LIN {X 0,Y 566.204,Z 705.957,A -85,B 0,C 180,E1 -2372.429,E2 -2372.429} C_VEL
LIN {X 0,Y 566.171,Z 705.961,A -85,B 0,C 180,E1 -2374.988,E2 -2374.988} C_VEL
LIN {X 0,Y 566.186,Z 705.954,A -85,B 0,C 180,E1 -2377.462,E2 -2377.462} C_VEL
LIN {X 0,Y 566.206,Z 705.952,A -85,B 0,C 180,E1 -2380.199,E2 -2380.199} C_VEL
LIN {X 0,Y 566.18,Z 705.961,A -85,B 0,C 180,E1 -2383.057,E2 -2383.057} C_VEL
LIN {X 0,Y 566.158,Z 705.957,A -85,B 0,C 180,E1 -2386.053,E2 -2386.053} C_VEL
LIN {X 0,Y 566.151,Z 705.966,A -85,B 0,C 180,E1 -2388.858,E2 -2388.858} C_VEL
LIN {X 0,Y 566.201,Z 705.955,A -85,B 0,C 180,E1 -2391.444,E2 -2391.444} C_VEL
LIN {X 0,Y 566.139,Z 705.959,A -85,B 0,C 180,E1 -2394.306,E2 -2394.306} C_VEL
LIN {X 0,Y 566.163,Z 705.963,A -85,B 0,C 180,E1 -2396.894,E2 -2396.894} C_VEL
LIN {X 0,Y 566.16,Z 705.963,A -85,B 0,C 180,E1 -2399.406,E2 -2399.406} C_VEL
LIN {X 0,Y 566.149,Z 705.959,A -85,B 0,C 180,E1 -2401.854,E2 -2401.854} C_VEL
LIN {X 0,Y 566.168,Z 705.955,A -85,B 0,C 180,E1 -2404.249,E2 -2404.249} C_VEL
LIN {X 0,Y 566.164,Z 705.964,A -85,B 0,C 180,E1 -2407.368,E2 -2407.368} C_VEL
LIN {X 0,Y 566.203,Z 705.956,A -85,B 0,C 180,E1 -2409.662,E2 -2409.662} C_VEL
LIN {X 0,Y 566.167,Z 705.958,A -85,B 0,C 180,E1 -2411.921,E2 -2411.921} C_VEL
LIN {X 0,Y 566.183,Z 705.956,A -85,B 0,C 180,E1 -2414.89,E2 -2414.89} C_VEL
LIN {X 0,Y 566.18,Z 705.959,A -85,B 0,C 180,E1 -2417.818,E2 -2417.818} C_VEL
LIN {X 0,Y 566.136,Z 705.962,A -85,B 0,C 180,E1 -2419.991,E2 -2419.991} C_VEL
LIN {X 0,Y 566.185,Z 705.955,A -85,B 0,C 180,E1 -2422.152,E2 -2422.152} C_VEL
LIN {X 0,Y 566.257,Z 705.946,A -85,B 0,C 180,E1 -2425.016,E2 -2425.016} C_VEL
LIN {X 0,Y 566.277,Z 705.948,A -85,B 0,C 180,E1 -2427.866,E2 -2427.866} C_VEL
LIN {X 0,Y 566.288,Z 705.945,A -85,B 0,C 180,E1 -2430,E2 -2430} C_VEL
LIN {X 0,Y 566.245,Z 705.945,A -85,B 0,C 180,E1 -2432.846,E2 -2432.846} C_VEL
LIN {X 0,Y 566.244,Z 705.955,A -85,B 0,C 180,E1 -2435.699,E2 -2435.699} C_VEL
LIN {X 0,Y 566.201,Z 705.952,A -85,B 0,C 180,E1 -2438.566,E2 -2438.566} C_VEL
LIN {X 0,Y 566.244,Z 705.949,A -85,B 0,C 180,E1 -2441.454,E2 -2441.454} C_VEL
LIN {X 0,Y 566.238,Z 705.948,A -85,B 0,C 180,E1 -2444.506,E2 -2444.506} C_VEL
LIN {X 0,Y 566.193,Z 705.953,A -85,B 0,C 180,E1 -2447.332,E2 -2447.332} C_VEL
LIN {X 0,Y 566.209,Z 705.955,A -85,B 0,C 180,E1 -2450.338,E2 -2450.338} C_VEL
LIN {X 0,Y 566.171,Z 705.955,A -85,B 0,C 180,E1 -2453.28,E2 -2453.28} C_VEL
LIN {X 0,Y 566.196,Z 705.955,A -85,B 0,C 180,E1 -2455.75,E2 -2455.75} C_VEL
LIN {X 0,Y 566.189,Z 705.962,A -85,B 0,C 180,E1 -2458.199,E2 -2458.199} C_VEL
LIN {X 0,Y 566.191,Z 705.952,A -85,B 0,C 180,E1 -2461.076,E2 -2461.076} C_VEL
LIN {X 0,Y 566.201,Z 705.953,A -85,B 0,C 180,E1 -2463.732,E2 -2463.732} C_VEL
LIN {X 0,Y 566.204,Z 705.957,A -85,B 0,C 180,E1 -2466.57,E2 -2466.57} C_VEL
LIN {X 0,Y 566.218,Z 705.949,A -85,B 0,C 180,E1 -2469.686,E2 -2469.686} C_VEL
LIN {X 0,Y 566.206,Z 705.953,A -85,B 0,C 180,E1 -2472.917,E2 -2472.917} C_VEL
LIN {X 0,Y 566.198,Z 705.954,A -85,B 0,C 180,E1 -2476.049,E2 -2476.049} C_VEL
LIN {X 0,Y 566.208,Z 705.953,A -85,B 0,C 180,E1 -2479.215,E2 -2479.215} C_VEL
LIN {X 0,Y 566.23,Z 706.075,A -85,B 0,C 180,E1 -2479.979,E2 -2479.979} C_VEL
LIN {X 0,Y 566.747,Z 710.218,A -85,B 0,C 180,E1 -2480.146,E2 -2480.146} C_VEL
LIN {X 0,Y 566.638,Z 721.443,A -85,B 0,C 180,E1 -2480.667,E2 -2480.667} C_VEL
LIN {X 0,Y 566.488,Z 730.938,A -85,B 0,C 180,E1 -2481.217,E2 -2481.217} C_VEL
LIN {X 0,Y 566.359,Z 740.262,A -85,B 0,C 180,E1 -2481.877,E2 -2481.877} C_VEL
LIN {X 0,Y 566.256,Z 749.282,A -85,B 0,C 180,E1 -2482.649,E2 -2482.649} C_VEL
LIN {X 0,Y 566.168,Z 756.903,A -85,B 0,C 180,E1 -2483.427,E2 -2483.427} C_VEL
LIN {X 0,Y 566.072,Z 764.081,A -85,B 0,C 180,E1 -2484.301,E2 -2484.301} C_VEL
LIN {X 0,Y 566.051,Z 770.069,A -85,B 0,C 180,E1 -2485.171,E2 -2485.171} C_VEL
LIN {X 0,Y 565.969,Z 775.031,A -85,B 0,C 180,E1 -2486.027,E2 -2486.027} C_VEL
LIN {X 0,Y 565.906,Z 779.166,A -85,B 0,C 180,E1 -2486.877,E2 -2486.877} C_VEL
LIN {X 0,Y 565.892,Z 782.518,A -85,B 0,C 180,E1 -2487.722,E2 -2487.722} C_VEL
LIN {X 0,Y 565.881,Z 786.273,A -85,B 0,C 180,E1 -2488.976,E2 -2488.976} C_VEL
LIN {X 0,Y 565.882,Z 788.867,A -85,B 0,C 180,E1 -2490.386,E2 -2490.386} C_VEL
LIN {X 0,Y 565.848,Z 789.586,A -85,B 0,C 180,E1 -2491.027,E2 -2491.027} C_VEL
LIN {X 0,Y 565.846,Z 789.967,A -85,B 0,C 180,E1 -2491.866,E2 -2491.866} C_VEL
LIN {X 0,Y 565.833,Z 789.805,A -85,B 0,C 180,E1 -2492.641,E2 -2492.641} C_VEL
LIN {X 0,Y 565.862,Z 789.206,A -85,B 0,C 180,E1 -2493.441,E2 -2493.441} C_VEL
LIN {X 0,Y 565.839,Z 788.123,A -85,B 0,C 180,E1 -2494.232,E2 -2494.232} C_VEL
LIN {X 0,Y 565.914,Z 785.462,A -85,B 0,C 180,E1 -2495.428,E2 -2495.428} C_VEL
LIN {X 0,Y 565.913,Z 781.702,A -85,B 0,C 180,E1 -2496.584,E2 -2496.584} C_VEL
LIN {X 0,Y 565.935,Z 776.65,A -85,B 0,C 180,E1 -2497.743,E2 -2497.743} C_VEL
LIN {X 0,Y 565.996,Z 771.822,A -85,B 0,C 180,E1 -2498.636,E2 -2498.636} C_VEL
LIN {X 0,Y 566.072,Z 765.057,A -85,B 0,C 180,E1 -2499.657,E2 -2499.657} C_VEL
LIN {X 0,Y 566.15,Z 759.073,A -85,B 0,C 180,E1 -2500.417,E2 -2500.417} C_VEL
LIN {X 0,Y 566.234,Z 752.096,A -85,B 0,C 180,E1 -2501.173,E2 -2501.173} C_VEL
LIN {X 0,Y 566.338,Z 742.679,A -85,B 0,C 180,E1 -2502.02,E2 -2502.02} C_VEL
LIN {X 0,Y 566.436,Z 733.894,A -85,B 0,C 180,E1 -2502.676,E2 -2502.676} C_VEL
LIN {X 0,Y 566.533,Z 724.261,A -85,B 0,C 180,E1 -2503.27,E2 -2503.27} C_VEL
LIN {X 0,Y 566.663,Z 713.636,A -85,B 0,C 180,E1 -2503.796,E2 -2503.796} C_VEL
LIN {X 0,Y 566.73,Z 708.105,A -85,B 0,C 180,E1 -2504.029,E2 -2504.029} C_VEL
LIN {X 0,Y 566.222,Z 705.951,A -85,B 0,C 180,E1 -2504.13,E2 -2504.13} C_VEL
LIN {X 0,Y 566.196,Z 705.953,A -85,B 0,C 180,E1 -2506.359,E2 -2506.359} C_VEL
LIN {X 0,Y 566.24,Z 705.947,A -85,B 0,C 180,E1 -2508.675,E2 -2508.675} C_VEL
LIN {X 0,Y 566.227,Z 705.955,A -85,B 0,C 180,E1 -2511.434,E2 -2511.434} C_VEL
LIN {X 0,Y 566.251,Z 705.946,A -85,B 0,C 180,E1 -2514.302,E2 -2514.302} C_VEL
LIN {X 0,Y 566.284,Z 705.95,A -85,B 0,C 180,E1 -2517.866,E2 -2517.866} C_VEL
LIN {X 0,Y 566.303,Z 705.938,A -85,B 0,C 180,E1 -2520.711,E2 -2520.711} C_VEL
LIN {X 0,Y 566.273,Z 705.941,A -85,B 0,C 180,E1 -2522.845,E2 -2522.845} C_VEL
LIN {X 0,Y 566.256,Z 705.95,A -85,B 0,C 180,E1 -2525.698,E2 -2525.698} C_VEL
LIN {X 0,Y 566.224,Z 705.956,A -85,B 0,C 180,E1 -2527.847,E2 -2527.847} C_VEL
LIN {X 0,Y 566.243,Z 705.946,A -85,B 0,C 180,E1 -2530.73,E2 -2530.73} C_VEL
LIN {X 0,Y 566.21,Z 705.95,A -85,B 0,C 180,E1 -2532.91,E2 -2532.91} C_VEL
LIN {X 0,Y 566.203,Z 705.949,A -85,B 0,C 180,E1 -2535.109,E2 -2535.109} C_VEL
LIN {X 0,Y 566.204,Z 705.951,A -85,B 0,C 180,E1 -2537.332,E2 -2537.332} C_VEL
LIN {X 0,Y 566.212,Z 705.956,A -85,B 0,C 180,E1 -2540.337,E2 -2540.337} C_VEL
LIN {X 0,Y 566.173,Z 705.954,A -85,B 0,C 180,E1 -2543.281,E2 -2543.281} C_VEL
LIN {X 0,Y 566.213,Z 705.951,A -85,B 0,C 180,E1 -2545.749,E2 -2545.749} C_VEL
LIN {X 0,Y 566.207,Z 705.958,A -85,B 0,C 180,E1 -2548.202,E2 -2548.202} C_VEL
LIN {X 0,Y 566.195,Z 705.952,A -85,B 0,C 180,E1 -2551.076,E2 -2551.076} C_VEL
LIN {X 0,Y 566.216,Z 705.95,A -85,B 0,C 180,E1 -2553.734,E2 -2553.734} C_VEL
LIN {X 0,Y 566.204,Z 705.96,A -85,B 0,C 180,E1 -2556.57,E2 -2556.57} C_VEL
LIN {X 0,Y 566.225,Z 705.95,A -85,B 0,C 180,E1 -2559.273,E2 -2559.273} C_VEL
LIN {X 0,Y 566.193,Z 705.955,A -85,B 0,C 180,E1 -2562.089,E2 -2562.089} C_VEL
LIN {X 0,Y 566.177,Z 705.959,A -85,B 0,C 180,E1 -2565.036,E2 -2565.036} C_VEL
LIN {X 0,Y 566.222,Z 705.952,A -85,B 0,C 180,E1 -2568.136,E2 -2568.136} C_VEL
LIN {X 0,Y 566.219,Z 705.96,A -85,B 0,C 180,E1 -2570.726,E2 -2570.726} C_VEL
LIN {X 0,Y 566.241,Z 706.07,A -85,B 0,C 180,E1 -2572.989,E2 -2572.989} C_VEL
LIN {X 0,Y 567.262,Z 712.594,A -85,B 0,C 180,E1 -2574.387,E2 -2574.387} C_VEL
LIN {X 0,Y 567.322,Z 727.831,A -85,B 0,C 180,E1 -2577.393,E2 -2577.393} C_VEL
LIN {X 0,Y 567.311,Z 742.969,A -85,B 0,C 180,E1 -2580.295,E2 -2580.295} C_VEL
LIN {X 0,Y 567.031,Z 758.624,A -85,B 0,C 180,E1 -2583.5,E2 -2583.5} C_VEL
LIN {X 0,Y 566.812,Z 772.321,A -85,B 0,C 180,E1 -2586.236,E2 -2586.236} C_VEL
LIN {X 0,Y 566.605,Z 787.97,A -85,B 0,C 180,E1 -2589.298,E2 -2589.298} C_VEL
LIN {X 0,Y 566.401,Z 803.622,A -85,B 0,C 180,E1 -2592.302,E2 -2592.302} C_VEL
LIN {X 0,Y 566.238,Z 819.258,A -85,B 0,C 180,E1 -2595.256,E2 -2595.256} C_VEL
LIN {X 0,Y 566.153,Z 830.11,A -85,B 0,C 180,E1 -2597.285,E2 -2597.285} C_VEL
LIN {X 0,Y 566.954,Z 837.081,A -85,B 0,C 180,E1 -2597.426,E2 -2597.426} C_VEL
LIN {X 0,Y 566.844,Z 850.733,A -85,B 0,C 180,E1 -2597.764,E2 -2597.764} C_VEL
LIN {X 0,Y 566.707,Z 863.522,A -85,B 0,C 180,E1 -2598.238,E2 -2598.238} C_VEL
LIN {X 0,Y 566.572,Z 875.723,A -85,B 0,C 180,E1 -2598.854,E2 -2598.854} C_VEL
LIN {X 0,Y 566.421,Z 886.478,A -85,B 0,C 180,E1 -2599.545,E2 -2599.545} C_VEL
LIN {X 0,Y 566.297,Z 896.645,A -85,B 0,C 180,E1 -2600.355,E2 -2600.355} C_VEL
LIN {X 0,Y 566.166,Z 905.786,A -85,B 0,C 180,E1 -2601.253,E2 -2601.253} C_VEL
LIN {X 0,Y 566.081,Z 914.689,A -85,B 0,C 180,E1 -2602.33,E2 -2602.33} C_VEL
LIN {X 0,Y 565.967,Z 921.955,A -85,B 0,C 180,E1 -2603.422,E2 -2603.422} C_VEL
LIN {X 0,Y 566.004,Z 926.68,A -85,B 0,C 180,E1 -2604.299,E2 -2604.299} C_VEL
LIN {X 0,Y 565.933,Z 931.371,A -85,B 0,C 180,E1 -2605.37,E2 -2605.37} C_VEL
LIN {X 0,Y 565.927,Z 934.957,A -85,B 0,C 180,E1 -2606.44,E2 -2606.44} C_VEL
LIN {X 0,Y 565.878,Z 936.808,A -85,B 0,C 180,E1 -2607.152,E2 -2607.152} C_VEL
LIN {X 0,Y 565.838,Z 938.199,A -85,B 0,C 180,E1 -2607.864,E2 -2607.864} C_VEL
LIN {X 0,Y 565.841,Z 939.785,A -85,B 0,C 180,E1 -2609.288,E2 -2609.288} C_VEL
LIN {X 0,Y 565.839,Z 940,A -85,B 0,C 180,E1 -2610,E2 -2610} C_VEL
LIN {X 0,Y 565.846,Z 939.186,A -85,B 0,C 180,E1 -2611.423,E2 -2611.423} C_VEL
LIN {X 0,Y 565.838,Z 938.2,A -85,B 0,C 180,E1 -2612.135,E2 -2612.135} C_VEL
LIN {X 0,Y 565.878,Z 936.81,A -85,B 0,C 180,E1 -2612.847,E2 -2612.847} C_VEL
LIN {X 0,Y 565.926,Z 933.896,A -85,B 0,C 180,E1 -2613.916,E2 -2613.916} C_VEL
LIN {X 0,Y 565.878,Z 929.949,A -85,B 0,C 180,E1 -2614.987,E2 -2614.987} C_VEL
LIN {X 0,Y 566.002,Z 924.867,A -85,B 0,C 180,E1 -2616.058,E2 -2616.058} C_VEL
LIN {X 0,Y 566.04,Z 918.469,A -85,B 0,C 180,E1 -2617.132,E2 -2617.132} C_VEL
LIN {X 0,Y 566.133,Z 910.479,A -85,B 0,C 180,E1 -2618.208,E2 -2618.208} C_VEL
LIN {X 0,Y 566.229,Z 902.337,A -85,B 0,C 180,E1 -2619.105,E2 -2619.105} C_VEL
LIN {X 0,Y 566.34,Z 892.402,A -85,B 0,C 180,E1 -2620.005,E2 -2620.005} C_VEL
LIN {X 0,Y 566.536,Z 881.306,A -85,B 0,C 180,E1 -2620.806,E2 -2620.806} C_VEL
LIN {X 0,Y 566.613,Z 870.179,A -85,B 0,C 180,E1 -2621.447,E2 -2621.447} C_VEL
LIN {X 0,Y 566.742,Z 857.987,A -85,B 0,C 180,E1 -2621.988,E2 -2621.988} C_VEL
LIN {X 0,Y 566.913,Z 845.178,A -85,B 0,C 180,E1 -2622.393,E2 -2622.393} C_VEL
LIN {X 0,Y 566.761,Z 833.946,A -85,B 0,C 180,E1 -2622.634,E2 -2622.634} C_VEL
LIN {X 0,Y 566.154,Z 830.034,A -85,B 0,C 180,E1 -2622.729,E2 -2622.729} C_VEL
LIN {X 0,Y 566.282,Z 815.361,A -85,B 0,C 180,E1 -2625.476,E2 -2625.476} C_VEL
LIN {X 0,Y 566.456,Z 799.71,A -85,B 0,C 180,E1 -2628.444,E2 -2628.444} C_VEL
LIN {X 0,Y 566.62,Z 784.878,A -85,B 0,C 180,E1 -2631.303,E2 -2631.303} C_VEL
LIN {X 0,Y 566.836,Z 770.363,A -85,B 0,C 180,E1 -2634.152,E2 -2634.152} C_VEL
LIN {X 0,Y 567.064,Z 756.117,A -85,B 0,C 180,E1 -2637.008,E2 -2637.008} C_VEL
LIN {X 0,Y 567.313,Z 742.161,A -85,B 0,C 180,E1 -2639.868,E2 -2639.868} C_VEL
LIN {X 0,Y 567.407,Z 727.53,A -85,B 0,C 180,E1 -2642.775,E2 -2642.775} C_VEL
LIN {X 0,Y 567.477,Z 715.115,A -85,B 0,C 180,E1 -2645.334,E2 -2645.334} C_VEL
LIN {X 0,Y 567.176,Z 710.471,A -85,B 0,C 180,E1 -2646.348,E2 -2646.348} C_VEL
LIN {X 0,Y 566.203,Z 705.96,A -85,B 0,C 180,E1 -2647.401,E2 -2647.401} C_VEL
LIN {X 0,Y 566.22,Z 705.951,A -85,B 0,C 180,E1 -2650.198,E2 -2650.198} C_VEL
LIN {X 0,Y 566.205,Z 705.958,A -85,B 0,C 180,E1 -2653.054,E2 -2653.054} C_VEL
LIN {X 0,Y 566.201,Z 705.952,A -85,B 0,C 180,E1 -2656.049,E2 -2656.049} C_VEL
LIN {X 0,Y 566.223,Z 705.956,A -85,B 0,C 180,E1 -2659.213,E2 -2659.213} C_VEL
LIN {X 0,Y 566.192,Z 705.959,A -85,B 0,C 180,E1 -2661.637,E2 -2661.637} C_VEL
LIN {X 0,Y 566.168,Z 705.955,A -85,B 0,C 180,E1 -2664.308,E2 -2664.308} C_VEL
LIN {X 0,Y 566.232,Z 705.948,A -85,B 0,C 180,E1 -2666.899,E2 -2666.899} C_VEL
LIN {X 0,Y 566.184,Z 705.96,A -85,B 0,C 180,E1 -2669.407,E2 -2669.407} C_VEL
LIN {X 0,Y 566.215,Z 705.955,A -85,B 0,C 180,E1 -2671.857,E2 -2671.857} C_VEL
LIN {X 0,Y 566.215,Z 705.951,A -85,B 0,C 180,E1 -2674.251,E2 -2674.251} C_VEL
LIN {X 0,Y 566.172,Z 705.954,A -85,B 0,C 180,E1 -2676.719,E2 -2676.719} C_VEL
LIN {X 0,Y 566.211,Z 705.958,A -85,B 0,C 180,E1 -2679.663,E2 -2679.663} C_VEL
LIN {X 0,Y 566.202,Z 705.951,A -85,B 0,C 180,E1 -2682.668,E2 -2682.668} C_VEL
LIN {X 0,Y 566.236,Z 705.953,A -85,B 0,C 180,E1 -2685.627,E2 -2685.627} C_VEL
LIN {X 0,Y 566.239,Z 705.947,A -85,B 0,C 180,E1 -2688.675,E2 -2688.675} C_VEL
LIN {X 0,Y 566.229,Z 705.95,A -85,B 0,C 180,E1 -2691.434,E2 -2691.434} C_VEL
LIN {X 0,Y 566.252,Z 705.95,A -85,B 0,C 180,E1 -2694.302,E2 -2694.302} C_VEL
LIN {X 0,Y 566.286,Z 705.947,A -85,B 0,C 180,E1 -2697.866,E2 -2697.866} C_VEL
LIN {X 0,Y 566.292,Z 705.941,A -85,B 0,C 180,E1 -2700.711,E2 -2700.711} C_VEL
LIN {X 0,Y 566.261,Z 705.945,A -85,B 0,C 180,E1 -2702.846,E2 -2702.846} C_VEL
LIN {X 0,Y 566.249,Z 705.948,A -85,B 0,C 180,E1 -2705.699,E2 -2705.699} C_VEL
LIN {X 0,Y 566.225,Z 705.953,A -85,B 0,C 180,E1 -2708.566,E2 -2708.566} C_VEL
LIN {X 0,Y 566.245,Z 705.946,A -85,B 0,C 180,E1 -2711.454,E2 -2711.454} C_VEL
LIN {X 0,Y 566.225,Z 705.956,A -85,B 0,C 180,E1 -2714.502,E2 -2714.502} C_VEL
LIN {X 0,Y 566.191,Z 705.952,A -85,B 0,C 180,E1 -2717.332,E2 -2717.332} C_VEL
LIN {X 0,Y 566.204,Z 705.951,A -85,B 0,C 180,E1 -2719.581,E2 -2719.581} C_VEL
LIN {X 0,Y 566.193,Z 705.953,A -85,B 0,C 180,E1 -2721.863,E2 -2721.863} C_VEL
LIN {X 0,Y 566.181,Z 705.957,A -85,B 0,C 180,E1 -2725.021,E2 -2725.021} C_VEL
LIN {X 0,Y 566.163,Z 705.956,A -85,B 0,C 180,E1 -2727.461,E2 -2727.461} C_VEL
LIN {X 0,Y 565.494,Z 706.042,A -85,B 0,C 180,E1 -2728.055,E2 -2728.055} C_VEL
LIN {X 0,Y 562.638,Z 706.399,A -85,B 0,C 180,E1 -2729.019,E2 -2729.019} C_VEL
LIN {X 0,Y 560.231,Z 706.698,A -85,B 0,C 180,E1 -2729.795,E2 -2729.795} C_VEL
LIN {X 0,Y 559.207,Z 706.829,A -85,B 0,C 180,E1 -2730.393,E2 -2730.393} C_VEL
LIN {X 0,Y 559.129,Z 706.834,A -85,B 0,C 180,E1 -2730.596,E2 -2730.596} C_VEL
LIN {X 0,Y 559.153,Z 706.838,A -85,B 0,C 180,E1 -2732.716,E2 -2732.716} C_VEL
LIN {X 0,Y 559.12,Z 706.835,A -85,B 0,C 180,E1 -2735.325,E2 -2735.325} C_VEL
LIN {X 0,Y 559.124,Z 706.833,A -85,B 0,C 180,E1 -2738.019,E2 -2738.019} C_VEL
LIN {X 0,Y 559.127,Z 706.841,A -85,B 0,C 180,E1 -2740.815,E2 -2740.815} C_VEL
LIN {X 0,Y 559.108,Z 706.835,A -85,B 0,C 180,E1 -2743.738,E2 -2743.738} C_VEL
LIN {X 0,Y 559.109,Z 706.836,A -85,B 0,C 180,E1 -2746.263,E2 -2746.263} C_VEL
LIN {X 0,Y 559.116,Z 706.841,A -85,B 0,C 180,E1 -2749.184,E2 -2749.184} C_VEL
LIN {X 0,Y 559.169,Z 706.835,A -85,B 0,C 180,E1 -2751.193,E2 -2751.193} C_VEL
LIN {X 0,Y 559.115,Z 706.835,A -85,B 0,C 180,E1 -2753.787,E2 -2753.787} C_VEL
LIN {X 0,Y 559.125,Z 706.834,A -85,B 0,C 180,E1 -2756.422,E2 -2756.422} C_VEL
LIN {X 0,Y 559.143,Z 706.838,A -85,B 0,C 180,E1 -2758.98,E2 -2758.98} C_VEL
LIN {X 0,Y 559.11,Z 706.838,A -85,B 0,C 180,E1 -2761.631,E2 -2761.631} C_VEL
LIN {X 0,Y 559.115,Z 706.835,A -85,B 0,C 180,E1 -2763.9,E2 -2763.9} C_VEL
LIN {X 0,Y 559.114,Z 706.841,A -85,B 0,C 180,E1 -2767.066,E2 -2767.066} C_VEL
LIN {X 0,Y 559.174,Z 706.835,A -85,B 0,C 180,E1 -2769.395,E2 -2769.395} C_VEL
LIN {X 0,Y 559.119,Z 706.839,A -85,B 0,C 180,E1 -2771.685,E2 -2771.685} C_VEL
LIN {X 0,Y 559.139,Z 706.833,A -85,B 0,C 180,E1 -2773.947,E2 -2773.947} C_VEL
LIN {X 0,Y 559.146,Z 706.831,A -85,B 0,C 180,E1 -2776.183,E2 -2776.183} C_VEL
LIN {X 0,Y 559.158,Z 706.833,A -85,B 0,C 180,E1 -2779.133,E2 -2779.133} C_VEL
LIN {X 0,Y 559.139,Z 706.834,A -85,B 0,C 180,E1 -2782.053,E2 -2782.053} C_VEL
LIN {X 0,Y 559.232,Z 706.821,A -85,B 0,C 180,E1 -2784.953,E2 -2784.953} C_VEL
LIN {X 0,Y 559.248,Z 706.824,A -85,B 0,C 180,E1 -2787.839,E2 -2787.839} C_VEL
LIN {X 0,Y 559.257,Z 706.821,A -85,B 0,C 180,E1 -2790,E2 -2790} C_VEL
LIN {X 0,Y 559.213,Z 706.822,A -85,B 0,C 180,E1 -2792.882,E2 -2792.882} C_VEL
LIN {X 0,Y 559.214,Z 706.831,A -85,B 0,C 180,E1 -2795.77,E2 -2795.77} C_VEL
LIN {X 0,Y 559.166,Z 706.828,A -85,B 0,C 180,E1 -2798.675,E2 -2798.675} C_VEL
LIN {X 0,Y 559.206,Z 706.828,A -85,B 0,C 180,E1 -2801.601,E2 -2801.601} C_VEL
LIN {X 0,Y 559.206,Z 706.824,A -85,B 0,C 180,E1 -2804.596,E2 -2804.596} C_VEL
LIN {X 0,Y 559.138,Z 706.834,A -85,B 0,C 180,E1 -2807.558,E2 -2807.558} C_VEL
LIN {X 0,Y 559.169,Z 706.834,A -85,B 0,C 180,E1 -2809.838,E2 -2809.838} C_VEL
LIN {X 0,Y 559.143,Z 706.839,A -85,B 0,C 180,E1 -2812.153,E2 -2812.153} C_VEL
LIN {X 0,Y 559.145,Z 706.83,A -85,B 0,C 180,E1 -2815.178,E2 -2815.178} C_VEL
LIN {X 0,Y 559.129,Z 706.835,A -85,B 0,C 180,E1 -2817.715,E2 -2817.715} C_VEL
LIN {X 0,Y 559.153,Z 706.839,A -85,B 0,C 180,E1 -2820.183,E2 -2820.183} C_VEL
LIN {X 0,Y 559.155,Z 706.832,A -85,B 0,C 180,E1 -2822.716,E2 -2822.716} C_VEL
LIN {X 0,Y 559.131,Z 706.831,A -85,B 0,C 180,E1 -2825.324,E2 -2825.324} C_VEL
LIN {X 0,Y 559.137,Z 706.835,A -85,B 0,C 180,E1 -2828.018,E2 -2828.018} C_VEL
LIN {X 0,Y 559.159,Z 706.831,A -85,B 0,C 180,E1 -2830.813,E2 -2830.813} C_VEL
LIN {X 0,Y 559.142,Z 706.83,A -85,B 0,C 180,E1 -2833.734,E2 -2833.734} C_VEL
LIN {X 0,Y 559.149,Z 706.836,A -85,B 0,C 180,E1 -2836.804,E2 -2836.804} C_VEL
LIN {X 0,Y 559.177,Z 706.829,A -85,B 0,C 180,E1 -2839.837,E2 -2839.837} C_VEL
LIN {X 0,Y 559.788,Z 710.922,A -85,B 0,C 180,E1 -2840.028,E2 -2840.028} C_VEL
LIN {X 0,Y 559.658,Z 721.465,A -85,B 0,C 180,E1 -2840.525,E2 -2840.525} C_VEL
LIN {X 0,Y 559.472,Z 732.021,A -85,B 0,C 180,E1 -2841.154,E2 -2841.154} C_VEL
LIN {X 0,Y 559.336,Z 740.517,A -85,B 0,C 180,E1 -2841.77,E2 -2841.77} C_VEL
LIN {X 0,Y 559.236,Z 748.955,A -85,B 0,C 180,E1 -2842.499,E2 -2842.499} C_VEL
LIN {X 0,Y 559.108,Z 756.352,A -85,B 0,C 180,E1 -2843.256,E2 -2843.256} C_VEL
LIN {X 0,Y 559.03,Z 762.612,A -85,B 0,C 180,E1 -2844.004,E2 -2844.004} C_VEL
LIN {X 0,Y 558.956,Z 769.522,A -85,B 0,C 180,E1 -2844.995,E2 -2844.995} C_VEL
LIN {X 0,Y 558.891,Z 774.491,A -85,B 0,C 180,E1 -2845.844,E2 -2845.844} C_VEL
LIN {X 0,Y 558.842,Z 779.251,A -85,B 0,C 180,E1 -2846.834,E2 -2846.834} C_VEL
LIN {X 0,Y 558.796,Z 783.939,A -85,B 0,C 180,E1 -2848.113,E2 -2848.113} C_VEL
LIN {X 0,Y 558.783,Z 786.313,A -85,B 0,C 180,E1 -2848.957,E2 -2848.957} C_VEL
LIN {X 0,Y 558.774,Z 788.662,A -85,B 0,C 180,E1 -2850.21,E2 -2850.21} C_VEL
LIN {X 0,Y 558.75,Z 789.905,A -85,B 0,C 180,E1 -2851.699,E2 -2851.699} C_VEL
LIN {X 0,Y 558.75,Z 789.585,A -85,B 0,C 180,E1 -2853.076,E2 -2853.076} C_VEL
LIN {X 0,Y 558.742,Z 788.659,A -85,B 0,C 180,E1 -2853.881,E2 -2853.881} C_VEL
LIN {X 0,Y 558.783,Z 786.806,A -85,B 0,C 180,E1 -2854.901,E2 -2854.901} C_VEL
LIN {X 0,Y 558.807,Z 784.25,A -85,B 0,C 180,E1 -2855.874,E2 -2855.874} C_VEL
LIN {X 0,Y 558.821,Z 780.058,A -85,B 0,C 180,E1 -2857.053,E2 -2857.053} C_VEL
LIN {X 0,Y 558.888,Z 774.655,A -85,B 0,C 180,E1 -2858.213,E2 -2858.213} C_VEL
LIN {X 0,Y 558.981,Z 767.676,A -85,B 0,C 180,E1 -2859.388,E2 -2859.388} C_VEL
LIN {X 0,Y 559.108,Z 759.09,A -85,B 0,C 180,E1 -2860.52,E2 -2860.52} C_VEL
LIN {X 0,Y 559.193,Z 751.891,A -85,B 0,C 180,E1 -2861.307,E2 -2861.307} C_VEL
LIN {X 0,Y 559.324,Z 743.595,A -85,B 0,C 180,E1 -2862.07,E2 -2862.07} C_VEL
LIN {X 0,Y 559.446,Z 733.913,A -85,B 0,C 180,E1 -2862.807,E2 -2862.807} C_VEL
LIN {X 0,Y 559.55,Z 724.513,A -85,B 0,C 180,E1 -2863.397,E2 -2863.397} C_VEL
LIN {X 0,Y 559.668,Z 715.312,A -85,B 0,C 180,E1 -2863.869,E2 -2863.869} C_VEL
LIN {X 0,Y 559.647,Z 708.978,A -85,B 0,C 180,E1 -2864.149,E2 -2864.149} C_VEL
LIN {X 0,Y 559.169,Z 706.83,A -85,B 0,C 180,E1 -2864.252,E2 -2864.252} C_VEL
LIN {X 0,Y 559.162,Z 706.83,A -85,B 0,C 180,E1 -2866.924,E2 -2866.924} C_VEL
LIN {X 0,Y 559.197,Z 706.828,A -85,B 0,C 180,E1 -2869.133,E2 -2869.133} C_VEL
LIN {X 0,Y 559.202,Z 706.827,A -85,B 0,C 180,E1 -2872.053,E2 -2872.053} C_VEL
LIN {X 0,Y 559.245,Z 706.818,A -85,B 0,C 180,E1 -2874.953,E2 -2874.953} C_VEL
LIN {X 0,Y 559.255,Z 706.826,A -85,B 0,C 180,E1 -2877.839,E2 -2877.839} C_VEL
LIN {X 0,Y 559.273,Z 706.814,A -85,B 0,C 180,E1 -2880.72,E2 -2880.72} C_VEL
LIN {X 0,Y 559.239,Z 706.817,A -85,B 0,C 180,E1 -2882.881,E2 -2882.881} C_VEL
LIN {X 0,Y 559.226,Z 706.827,A -85,B 0,C 180,E1 -2885.77,E2 -2885.77} C_VEL
LIN {X 0,Y 559.174,Z 706.826,A -85,B 0,C 180,E1 -2888.675,E2 -2888.675} C_VEL
LIN {X 0,Y 559.21,Z 706.825,A -85,B 0,C 180,E1 -2891.6,E2 -2891.6} C_VEL
LIN {X 0,Y 559.205,Z 706.823,A -85,B 0,C 180,E1 -2894.595,E2 -2894.595} C_VEL
LIN {X 0,Y 559.147,Z 706.831,A -85,B 0,C 180,E1 -2897.557,E2 -2897.557} C_VEL
LIN {X 0,Y 559.171,Z 706.831,A -85,B 0,C 180,E1 -2899.837,E2 -2899.837} C_VEL
LIN {X 0,Y 559.145,Z 706.838,A -85,B 0,C 180,E1 -2902.153,E2 -2902.153} C_VEL
LIN {X 0,Y 559.179,Z 706.826,A -85,B 0,C 180,E1 -2905.298,E2 -2905.298} C_VEL
LIN {X 0,Y 559.161,Z 706.829,A -85,B 0,C 180,E1 -2907.713,E2 -2907.713} C_VEL
LIN {X 0,Y 559.157,Z 706.835,A -85,B 0,C 180,E1 -2910.183,E2 -2910.183} C_VEL
LIN {X 0,Y 559.179,Z 706.831,A -85,B 0,C 180,E1 -2912.714,E2 -2912.714} C_VEL
LIN {X 0,Y 559.134,Z 706.832,A -85,B 0,C 180,E1 -2915.324,E2 -2915.324} C_VEL
LIN {X 0,Y 559.138,Z 706.834,A -85,B 0,C 180,E1 -2918.017,E2 -2918.017} C_VEL
LIN {X 0,Y 559.177,Z 706.833,A -85,B 0,C 180,E1 -2920.811,E2 -2920.811} C_VEL
LIN {X 0,Y 559.145,Z 706.831,A -85,B 0,C 180,E1 -2923.734,E2 -2923.734} C_VEL
LIN {X 0,Y 559.169,Z 706.837,A -85,B 0,C 180,E1 -2926.801,E2 -2926.801} C_VEL
LIN {X 0,Y 559.166,Z 706.835,A -85,B 0,C 180,E1 -2929.188,E2 -2929.188} C_VEL
LIN {X 0,Y 559.137,Z 706.837,A -85,B 0,C 180,E1 -2931.982,E2 -2931.982} C_VEL
LIN {X 0,Y 559.198,Z 706.945,A -85,B 0,C 180,E1 -2932.798,E2 -2932.798} C_VEL
LIN {X 0,Y 560.308,Z 713.782,A -85,B 0,C 180,E1 -2934.287,E2 -2934.287} C_VEL
LIN {X 0,Y 560.332,Z 729.084,A -85,B 0,C 180,E1 -2937.362,E2 -2937.362} C_VEL
LIN {X 0,Y 560.32,Z 743.41,A -85,B 0,C 180,E1 -2940.13,E2 -2940.13} C_VEL
LIN {X 0,Y 560.217,Z 752.754,A -85,B 0,C 180,E1 -2941.937,E2 -2941.937} C_VEL
LIN {X 0,Y 559.994,Z 766.449,A -85,B 0,C 180,E1 -2944.741,E2 -2944.741} C_VEL
LIN {X 0,Y 559.741,Z 780.144,A -85,B 0,C 180,E1 -2947.483,E2 -2947.483} C_VEL
LIN {X 0,Y 559.514,Z 795.003,A -85,B 0,C 180,E1 -2950.402,E2 -2950.402} C_VEL
LIN {X 0,Y 559.329,Z 809.491,A -85,B 0,C 180,E1 -2953.202,E2 -2953.202} C_VEL
LIN {X 0,Y 559.173,Z 825.142,A -85,B 0,C 180,E1 -2956.184,E2 -2956.184} C_VEL
LIN {X 0,Y 559.103,Z 830.156,A -85,B 0,C 180,E1 -2957.131,E2 -2957.131} C_VEL
LIN {X 0,Y 560.027,Z 837.081,A -85,B 0,C 180,E1 -2957.267,E2 -2957.267} C_VEL
LIN {X 0,Y 559.91,Z 850.734,A -85,B 0,C 180,E1 -2957.61,E2 -2957.61} C_VEL
LIN {X 0,Y 559.77,Z 863.521,A -85,B 0,C 180,E1 -2958.09,E2 -2958.09} C_VEL
LIN {X 0,Y 559.604,Z 876.209,A -85,B 0,C 180,E1 -2958.742,E2 -2958.742} C_VEL
LIN {X 0,Y 559.408,Z 887.745,A -85,B 0,C 180,E1 -2959.504,E2 -2959.504} C_VEL
LIN {X 0,Y 559.241,Z 898.6,A -85,B 0,C 180,E1 -2960.415,E2 -2960.415} C_VEL
LIN {X 0,Y 559.127,Z 907.412,A -85,B 0,C 180,E1 -2961.325,E2 -2961.325} C_VEL
LIN {X 0,Y 558.996,Z 916,A -85,B 0,C 180,E1 -2962.414,E2 -2962.414} C_VEL
LIN {X 0,Y 558.885,Z 923.688,A -85,B 0,C 180,E1 -2963.649,E2 -2963.649} C_VEL
LIN {X 0,Y 558.869,Z 928.365,A -85,B 0,C 180,E1 -2964.588,E2 -2964.588} C_VEL
LIN {X 0,Y 558.868,Z 932.677,A -85,B 0,C 180,E1 -2965.673,E2 -2965.673} C_VEL
LIN {X 0,Y 558.836,Z 934.957,A -85,B 0,C 180,E1 -2966.395,E2 -2966.395} C_VEL
LIN {X 0,Y 558.799,Z 936.808,A -85,B 0,C 180,E1 -2967.116,E2 -2967.116} C_VEL
LIN {X 0,Y 558.745,Z 939.185,A -85,B 0,C 180,E1 -2968.558,E2 -2968.558} C_VEL
LIN {X 0,Y 558.74,Z 940,A -85,B 0,C 180,E1 -2970,E2 -2970} C_VEL
LIN {X 0,Y 558.745,Z 939.186,A -85,B 0,C 180,E1 -2971.441,E2 -2971.441} C_VEL
LIN {X 0,Y 558.799,Z 936.81,A -85,B 0,C 180,E1 -2972.884,E2 -2972.884} C_VEL
LIN {X 0,Y 558.844,Z 933.896,A -85,B 0,C 180,E1 -2973.966,E2 -2973.966} C_VEL
LIN {X 0,Y 558.798,Z 929.949,A -85,B 0,C 180,E1 -2975.051,E2 -2975.051} C_VEL
LIN {X 0,Y 558.921,Z 924.867,A -85,B 0,C 180,E1 -2976.135,E2 -2976.135} C_VEL
LIN {X 0,Y 558.977,Z 918.469,A -85,B 0,C 180,E1 -2977.223,E2 -2977.223} C_VEL
LIN {X 0,Y 559.099,Z 910.479,A -85,B 0,C 180,E1 -2978.312,E2 -2978.312} C_VEL
LIN {X 0,Y 559.195,Z 902.336,A -85,B 0,C 180,E1 -2979.221,E2 -2979.221} C_VEL
LIN {X 0,Y 559.351,Z 892.402,A -85,B 0,C 180,E1 -2980.131,E2 -2980.131} C_VEL
LIN {X 0,Y 559.543,Z 881.404,A -85,B 0,C 180,E1 -2980.936,E2 -2980.936} C_VEL
LIN {X 0,Y 559.671,Z 869.464,A -85,B 0,C 180,E1 -2981.628,E2 -2981.628} C_VEL
LIN {X 0,Y 559.824,Z 856.767,A -85,B 0,C 180,E1 -2982.185,E2 -2982.185} C_VEL
LIN {X 0,Y 559.988,Z 843.349,A -85,B 0,C 180,E1 -2982.595,E2 -2982.595} C_VEL
LIN {X 0,Y 559.822,Z 834.611,A -85,B 0,C 180,E1 -2982.783,E2 -2982.783} C_VEL
LIN {X 0,Y 559.112,Z 830.034,A -85,B 0,C 180,E1 -2982.892,E2 -2982.892} C_VEL
LIN {X 0,Y 559.254,Z 815.361,A -85,B 0,C 180,E1 -2985.675,E2 -2985.675} C_VEL
LIN {X 0,Y 559.424,Z 801.666,A -85,B 0,C 180,E1 -2988.305,E2 -2988.305} C_VEL
LIN {X 0,Y 559.636,Z 787.971,A -85,B 0,C 180,E1 -2990.972,E2 -2990.972} C_VEL
LIN {X 0,Y 559.843,Z 774.276,A -85,B 0,C 180,E1 -2993.685,E2 -2993.685} C_VEL
LIN {X 0,Y 560.106,Z 760.581,A -85,B 0,C 180,E1 -2996.452,E2 -2996.452} C_VEL
LIN {X 0,Y 560.298,Z 746.652,A -85,B 0,C 180,E1 -2999.287,E2 -2999.287} C_VEL
LIN {X 0,Y 560.418,Z 734.158,A -85,B 0,C 180,E1 -3001.783,E2 -3001.783} C_VEL
LIN {X 0,Y 560.552,Z 720.629,A -85,B 0,C 180,E1 -3004.564,E2 -3004.564} C_VEL
LIN {X 0,Y 560.495,Z 713.436,A -85,B 0,C 180,E1 -3006.109,E2 -3006.109} C_VEL
LIN {X 0,Y 559.15,Z 706.838,A -85,B 0,C 180,E1 -3007.689,E2 -3007.689} C_VEL
LIN {X 0,Y 559.165,Z 706.831,A -85,B 0,C 180,E1 -3009.942,E2 -3009.942} C_VEL
LIN {X 0,Y 559.165,Z 706.831,A -85,B 0,C 180,E1 -3012.743,E2 -3012.743} C_VEL
LIN {X 0,Y 559.156,Z 706.832,A -85,B 0,C 180,E1 -3015.761,E2 -3015.761} C_VEL
LIN {X 0,Y 559.169,Z 706.827,A -85,B 0,C 180,E1 -3018.23,E2 -3018.23} C_VEL
LIN {X 0,Y 559.18,Z 706.831,A -85,B 0,C 180,E1 -3021.191,E2 -3021.191} C_VEL
LIN {X 0,Y 559.143,Z 706.835,A -85,B 0,C 180,E1 -3023.789,E2 -3023.789} C_VEL
LIN {X 0,Y 559.168,Z 706.827,A -85,B 0,C 180,E1 -3026.425,E2 -3026.425} C_VEL
LIN {X 0,Y 559.158,Z 706.83,A -85,B 0,C 180,E1 -3028.981,E2 -3028.981} C_VEL
LIN {X 0,Y 559.171,Z 706.836,A -85,B 0,C 180,E1 -3031.619,E2 -3031.619} C_VEL
LIN {X 0,Y 559.182,Z 706.831,A -85,B 0,C 180,E1 -3033.903,E2 -3033.903} C_VEL
LIN {X 0,Y 559.141,Z 706.83,A -85,B 0,C 180,E1 -3036.572,E2 -3036.572} C_VEL
LIN {X 0,Y 559.18,Z 706.83,A -85,B 0,C 180,E1 -3039.395,E2 -3039.395} C_VEL
LIN {X 0,Y 559.145,Z 706.838,A -85,B 0,C 180,E1 -3041.686,E2 -3041.686} C_VEL
LIN {X 0,Y 559.168,Z 706.836,A -85,B 0,C 180,E1 -3043.948,E2 -3043.948} C_VEL
LIN {X 0,Y 559.171,Z 706.832,A -85,B 0,C 180,E1 -3046.184,E2 -3046.184} C_VEL
LIN {X 0,Y 559.198,Z 706.824,A -85,B 0,C 180,E1 -3049.134,E2 -3049.134} C_VEL
LIN {X 0,Y 559.202,Z 706.832,A -85,B 0,C 180,E1 -3052.054,E2 -3052.054} C_VEL
LIN {X 0,Y 559.252,Z 706.817,A -85,B 0,C 180,E1 -3054.953,E2 -3054.953} C_VEL
LIN {X 0,Y 559.257,Z 706.822,A -85,B 0,C 180,E1 -3057.84,E2 -3057.84} C_VEL
LIN {X 0,Y 559.264,Z 706.817,A -85,B 0,C 180,E1 -3060.72,E2 -3060.72} C_VEL
LIN {X 0,Y 559.229,Z 706.82,A -85,B 0,C 180,E1 -3062.882,E2 -3062.882} C_VEL
LIN {X 0,Y 559.218,Z 706.824,A -85,B 0,C 180,E1 -3065.77,E2 -3065.77} C_VEL
LIN {X 0,Y 559.183,Z 706.829,A -85,B 0,C 180,E1 -3068.675,E2 -3068.675} C_VEL
LIN {X 0,Y 559.208,Z 706.823,A -85,B 0,C 180,E1 -3071.601,E2 -3071.601} C_VEL
LIN {X 0,Y 559.184,Z 706.832,A -85,B 0,C 180,E1 -3074.588,E2 -3074.588} C_VEL
LIN {X 0,Y 559.136,Z 706.832,A -85,B 0,C 180,E1 -3077.558,E2 -3077.558} C_VEL
LIN {X 0,Y 559.167,Z 706.829,A -85,B 0,C 180,E1 -3079.838,E2 -3079.838} C_VEL
LIN {X 0,Y 559.141,Z 706.835,A -85,B 0,C 180,E1 -3082.153,E2 -3082.153} C_VEL
LIN {X 0,Y 559.14,Z 706.832,A -85,B 0,C 180,E1 -3085.178,E2 -3085.178} C_VEL
LIN {X 0,Y 559.136,Z 706.838,A -85,B 0,C 180,E1 -3088.374,E2 -3088.374} C_VEL
LIN {X 0,Y 559.129,Z 706.834,A -85,B 0,C 180,E1 -3090.596,E2 -3090.596} C_VEL
LIN {X 0,Y 558.472,Z 706.918,A -85,B 0,C 180,E1 -3091.198,E2 -3091.198} C_VEL
LIN {X 0,Y 555.613,Z 707.273,A -85,B 0,C 180,E1 -3092.174,E2 -3092.174} C_VEL
LIN {X 0,Y 553.196,Z 707.577,A -85,B 0,C 180,E1 -3092.96,E2 -3092.96} C_VEL
LIN {X 0,Y 552.167,Z 707.7,A -85,B 0,C 180,E1 -3093.566,E2 -3093.566} C_VEL
LIN {X 0,Y 552.089,Z 707.709,A -85,B 0,C 180,E1 -3093.772,E2 -3093.772} C_VEL
LIN {X 0,Y 552.098,Z 707.716,A -85,B 0,C 180,E1 -3096.748,E2 -3096.748} C_VEL
LIN {X 0,Y 552.11,Z 707.708,A -85,B 0,C 180,E1 -3099.529,E2 -3099.529} C_VEL
LIN {X 0,Y 552.085,Z 707.713,A -85,B 0,C 180,E1 -3102.43,E2 -3102.43} C_VEL
LIN {X 0,Y 552.076,Z 707.712,A -85,B 0,C 180,E1 -3105.56,E2 -3105.56} C_VEL
LIN {X 0,Y 552.06,Z 707.717,A -85,B 0,C 180,E1 -3108.548,E2 -3108.548} C_VEL
LIN {X 0,Y 552.112,Z 707.711,A -85,B 0,C 180,E1 -3111.41,E2 -3111.41} C_VEL
LIN {X 0,Y 552.064,Z 707.715,A -85,B 0,C 180,E1 -3114.563,E2 -3114.563} C_VEL
LIN {X 0,Y 552.097,Z 707.716,A -85,B 0,C 180,E1 -3117.157,E2 -3117.157} C_VEL
LIN {X 0,Y 552.077,Z 707.711,A -85,B 0,C 180,E1 -3119.957,E2 -3119.957} C_VEL
LIN {X 0,Y 552.077,Z 707.718,A -85,B 0,C 180,E1 -3123.014,E2 -3123.014} C_VEL
LIN {X 0,Y 552.07,Z 707.713,A -85,B 0,C 180,E1 -3125.96,E2 -3125.96} C_VEL
LIN {X 0,Y 552.112,Z 707.707,A -85,B 0,C 180,E1 -3128.337,E2 -3128.337} C_VEL
LIN {X 0,Y 552.151,Z 707.703,A -85,B 0,C 180,E1 -3130.674,E2 -3130.674} C_VEL
LIN {X 0,Y 552.087,Z 707.714,A -85,B 0,C 180,E1 -3133.736,E2 -3133.736} C_VEL
LIN {X 0,Y 552.114,Z 707.708,A -85,B 0,C 180,E1 -3136.004,E2 -3136.004} C_VEL
LIN {X 0,Y 552.127,Z 707.707,A -85,B 0,C 180,E1 -3138.993,E2 -3138.993} C_VEL
LIN {X 0,Y 552.109,Z 707.711,A -85,B 0,C 180,E1 -3141.951,E2 -3141.951} C_VEL
LIN {X 0,Y 552.207,Z 707.695,A -85,B 0,C 180,E1 -3144.889,E2 -3144.889} C_VEL
LIN {X 0,Y 552.22,Z 707.7,A -85,B 0,C 180,E1 -3147.812,E2 -3147.812} C_VEL
LIN {X 0,Y 552.225,Z 707.697,A -85,B 0,C 180,E1 -3150,E2 -3150} C_VEL
LIN {X 0,Y 552.181,Z 707.698,A -85,B 0,C 180,E1 -3152.918,E2 -3152.918} C_VEL
LIN {X 0,Y 552.185,Z 707.705,A -85,B 0,C 180,E1 -3155.844,E2 -3155.844} C_VEL
LIN {X 0,Y 552.137,Z 707.703,A -85,B 0,C 180,E1 -3158.786,E2 -3158.786} C_VEL
LIN {X 0,Y 552.162,Z 707.708,A -85,B 0,C 180,E1 -3161.751,E2 -3161.751} C_VEL
LIN {X 0,Y 552.14,Z 707.703,A -85,B 0,C 180,E1 -3164.748,E2 -3164.748} C_VEL
LIN {X 0,Y 552.097,Z 707.714,A -85,B 0,C 180,E1 -3167.789,E2 -3167.789} C_VEL
LIN {X 0,Y 552.13,Z 707.712,A -85,B 0,C 180,E1 -3170.101,E2 -3170.101} C_VEL
LIN {X 0,Y 552.094,Z 707.713,A -85,B 0,C 180,E1 -3172.451,E2 -3172.451} C_VEL
LIN {X 0,Y 552.089,Z 707.709,A -85,B 0,C 180,E1 -3175.335,E2 -3175.335} C_VEL
LIN {X 0,Y 552.081,Z 707.719,A -85,B 0,C 180,E1 -3178.1,E2 -3178.1} C_VEL
LIN {X 0,Y 552.103,Z 707.711,A -85,B 0,C 180,E1 -3180.61,E2 -3180.61} C_VEL
LIN {X 0,Y 552.11,Z 707.706,A -85,B 0,C 180,E1 -3183.187,E2 -3183.187} C_VEL
LIN {X 0,Y 552.089,Z 707.711,A -85,B 0,C 180,E1 -3185.844,E2 -3185.844} C_VEL
LIN {X 0,Y 552.121,Z 707.711,A -85,B 0,C 180,E1 -3188.589,E2 -3188.589} C_VEL
LIN {X 0,Y 552.124,Z 707.704,A -85,B 0,C 180,E1 -3191.446,E2 -3191.446} C_VEL
LIN {X 0,Y 552.093,Z 707.718,A -85,B 0,C 180,E1 -3194.531,E2 -3194.531} C_VEL
LIN {X 0,Y 552.134,Z 707.704,A -85,B 0,C 180,E1 -3197.585,E2 -3197.585} C_VEL
LIN {X 0,Y 552.129,Z 707.706,A -85,B 0,C 180,E1 -3199.725,E2 -3199.725} C_VEL
LIN {X 0,Y 552.834,Z 710.917,A -85,B 0,C 180,E1 -3199.875,E2 -3199.875} C_VEL
LIN {X 0,Y 552.672,Z 721.851,A -85,B 0,C 180,E1 -3200.401,E2 -3200.401} C_VEL
LIN {X 0,Y 552.521,Z 731.068,A -85,B 0,C 180,E1 -3200.951,E2 -3200.951} C_VEL
LIN {X 0,Y 552.342,Z 740.188,A -85,B 0,C 180,E1 -3201.612,E2 -3201.612} C_VEL
LIN {X 0,Y 552.208,Z 748.619,A -85,B 0,C 180,E1 -3202.345,E2 -3202.345} C_VEL
LIN {X 0,Y 552.088,Z 755.309,A -85,B 0,C 180,E1 -3203.023,E2 -3203.023} C_VEL
LIN {X 0,Y 551.959,Z 762.755,A -85,B 0,C 180,E1 -3203.921,E2 -3203.921} C_VEL
LIN {X 0,Y 551.881,Z 768.941,A -85,B 0,C 180,E1 -3204.809,E2 -3204.809} C_VEL
LIN {X 0,Y 551.793,Z 775.228,A -85,B 0,C 180,E1 -3205.915,E2 -3205.915} C_VEL
LIN {X 0,Y 551.747,Z 779.328,A -85,B 0,C 180,E1 -3206.789,E2 -3206.789} C_VEL
LIN {X 0,Y 551.724,Z 782.676,A -85,B 0,C 180,E1 -3207.655,E2 -3207.655} C_VEL
LIN {X 0,Y 551.733,Z 785.499,A -85,B 0,C 180,E1 -3208.589,E2 -3208.589} C_VEL
LIN {X 0,Y 551.694,Z 788.451,A -85,B 0,C 180,E1 -3210.026,E2 -3210.026} C_VEL
LIN {X 0,Y 551.651,Z 789.615,A -85,B 0,C 180,E1 -3211.045,E2 -3211.045} C_VEL
LIN {X 0,Y 551.666,Z 789.97,A -85,B 0,C 180,E1 -3211.877,E2 -3211.877} C_VEL
LIN {X 0,Y 551.652,Z 789.578,A -85,B 0,C 180,E1 -3213.1,E2 -3213.1} C_VEL
LIN {X 0,Y 551.644,Z 788.05,A -85,B 0,C 180,E1 -3214.331,E2 -3214.331} C_VEL
LIN {X 0,Y 551.733,Z 785.37,A -85,B 0,C 180,E1 -3215.544,E2 -3215.544} C_VEL
LIN {X 0,Y 551.75,Z 781.527,A -85,B 0,C 180,E1 -3216.742,E2 -3216.742} C_VEL
LIN {X 0,Y 551.779,Z 778.35,A -85,B 0,C 180,E1 -3217.535,E2 -3217.535} C_VEL
LIN {X 0,Y 551.839,Z 772.122,A -85,B 0,C 180,E1 -3218.753,E2 -3218.753} C_VEL
LIN {X 0,Y 551.93,Z 766.17,A -85,B 0,C 180,E1 -3219.697,E2 -3219.697} C_VEL
LIN {X 0,Y 552.045,Z 758.724,A -85,B 0,C 180,E1 -3220.67,E2 -3220.67} C_VEL
LIN {X 0,Y 552.154,Z 751.688,A -85,B 0,C 180,E1 -3221.445,E2 -3221.445} C_VEL
LIN {X 0,Y 552.31,Z 743.349,A -85,B 0,C 180,E1 -3222.218,E2 -3222.218} C_VEL
LIN {X 0,Y 552.441,Z 734.772,A -85,B 0,C 180,E1 -3222.885,E2 -3222.885} C_VEL
LIN {X 0,Y 552.554,Z 725.851,A -85,B 0,C 180,E1 -3223.465,E2 -3223.465} C_VEL
LIN {X 0,Y 552.696,Z 715.918,A -85,B 0,C 180,E1 -3223.992,E2 -3223.992} C_VEL
LIN {X 0,Y 552.771,Z 710.612,A -85,B 0,C 180,E1 -3224.231,E2 -3224.231} C_VEL
LIN {X 0,Y 552.121,Z 707.707,A -85,B 0,C 180,E1 -3224.377,E2 -3224.377} C_VEL
LIN {X 0,Y 552.124,Z 707.706,A -85,B 0,C 180,E1 -3226.754,E2 -3226.754} C_VEL
LIN {X 0,Y 552.165,Z 707.703,A -85,B 0,C 180,E1 -3228.993,E2 -3228.993} C_VEL
LIN {X 0,Y 552.157,Z 707.706,A -85,B 0,C 180,E1 -3231.951,E2 -3231.951} C_VEL
LIN {X 0,Y 552.22,Z 707.693,A -85,B 0,C 180,E1 -3234.889,E2 -3234.889} C_VEL
LIN {X 0,Y 552.226,Z 707.702,A -85,B 0,C 180,E1 -3237.812,E2 -3237.812} C_VEL
LIN {X 0,Y 552.243,Z 707.689,A -85,B 0,C 180,E1 -3240.729,E2 -3240.729} C_VEL
LIN {X 0,Y 552.206,Z 707.693,A -85,B 0,C 180,E1 -3242.918,E2 -3242.918} C_VEL
LIN {X 0,Y 552.198,Z 707.704,A -85,B 0,C 180,E1 -3245.844,E2 -3245.844} C_VEL
LIN {X 0,Y 552.145,Z 707.7,A -85,B 0,C 180,E1 -3248.786,E2 -3248.786} C_VEL
LIN {X 0,Y 552.167,Z 707.704,A -85,B 0,C 180,E1 -3251.75,E2 -3251.75} C_VEL
LIN {X 0,Y 552.141,Z 707.702,A -85,B 0,C 180,E1 -3254.748,E2 -3254.748} C_VEL
LIN {X 0,Y 552.104,Z 707.711,A -85,B 0,C 180,E1 -3257.789,E2 -3257.789} C_VEL
LIN {X 0,Y 552.131,Z 707.712,A -85,B 0,C 180,E1 -3260.101,E2 -3260.101} C_VEL
LIN {X 0,Y 552.096,Z 707.714,A -85,B 0,C 180,E1 -3262.451,E2 -3262.451} C_VEL
LIN {X 0,Y 552.159,Z 707.7,A -85,B 0,C 180,E1 -3265.35,E2 -3265.35} C_VEL
LIN {X 0,Y 552.114,Z 707.712,A -85,B 0,C 180,E1 -3268.098,E2 -3268.098} C_VEL
LIN {X 0,Y 552.107,Z 707.713,A -85,B 0,C 180,E1 -3270.609,E2 -3270.609} C_VEL
LIN {X 0,Y 552.127,Z 707.705,A -85,B 0,C 180,E1 -3273.185,E2 -3273.185} C_VEL
LIN {X 0,Y 552.091,Z 707.711,A -85,B 0,C 180,E1 -3275.843,E2 -3275.843} C_VEL
LIN {X 0,Y 552.129,Z 707.708,A -85,B 0,C 180,E1 -3279.062,E2 -3279.062} C_VEL
LIN {X 0,Y 552.132,Z 707.705,A -85,B 0,C 180,E1 -3281.445,E2 -3281.445} C_VEL
LIN {X 0,Y 552.099,Z 707.717,A -85,B 0,C 180,E1 -3284.532,E2 -3284.532} C_VEL
LIN {X 0,Y 552.135,Z 707.706,A -85,B 0,C 180,E1 -3287.584,E2 -3287.584} C_VEL
LIN {X 0,Y 552.134,Z 707.713,A -85,B 0,C 180,E1 -3290.473,E2 -3290.473} C_VEL
LIN {X 0,Y 552.146,Z 707.835,A -85,B 0,C 180,E1 -3292.599,E2 -3292.599} C_VEL
LIN {X 0,Y 553.318,Z 714.214,A -85,B 0,C 180,E1 -3294.024,E2 -3294.024} C_VEL
LIN {X 0,Y 553.349,Z 727.103,A -85,B 0,C 180,E1 -3296.68,E2 -3296.68} C_VEL
LIN {X 0,Y 553.304,Z 742.575,A -85,B 0,C 180,E1 -3299.738,E2 -3299.738} C_VEL
LIN {X 0,Y 553.209,Z 758.591,A -85,B 0,C 180,E1 -3302.784,E2 -3302.784} C_VEL
LIN {X 0,Y 552.943,Z 772.319,A -85,B 0,C 180,E1 -3305.601,E2 -3305.601} C_VEL
LIN {X 0,Y 552.67,Z 786.014,A -85,B 0,C 180,E1 -3308.36,E2 -3308.36} C_VEL
LIN {X 0,Y 552.446,Z 799.709,A -85,B 0,C 180,E1 -3311.071,E2 -3311.071} C_VEL
LIN {X 0,Y 552.274,Z 813.404,A -85,B 0,C 180,E1 -3313.742,E2 -3313.742} C_VEL
LIN {X 0,Y 552.06,Z 829.055,A -85,B 0,C 180,E1 -3316.753,E2 -3316.753} C_VEL
LIN {X 0,Y 552.072,Z 830.156,A -85,B 0,C 180,E1 -3316.964,E2 -3316.964} C_VEL
LIN {X 0,Y 553.111,Z 838.222,A -85,B 0,C 180,E1 -3317.129,E2 -3317.129} C_VEL
LIN {X 0,Y 552.973,Z 851.494,A -85,B 0,C 180,E1 -3317.475,E2 -3317.475} C_VEL
LIN {X 0,Y 552.818,Z 863.512,A -85,B 0,C 180,E1 -3317.938,E2 -3317.938} C_VEL
LIN {X 0,Y 552.656,Z 875.819,A -85,B 0,C 180,E1 -3318.575,E2 -3318.575} C_VEL
LIN {X 0,Y 552.462,Z 886.48,A -85,B 0,C 180,E1 -3319.278,E2 -3319.278} C_VEL
LIN {X 0,Y 552.277,Z 896.645,A -85,B 0,C 180,E1 -3320.108,E2 -3320.108} C_VEL
LIN {X 0,Y 552.104,Z 905.785,A -85,B 0,C 180,E1 -3321.029,E2 -3321.029} C_VEL
LIN {X 0,Y 551.96,Z 914.688,A -85,B 0,C 180,E1 -3322.133,E2 -3322.133} C_VEL
LIN {X 0,Y 551.835,Z 921.848,A -85,B 0,C 180,E1 -3323.234,E2 -3323.234} C_VEL
LIN {X 0,Y 551.804,Z 928.365,A -85,B 0,C 180,E1 -3324.518,E2 -3324.518} C_VEL
LIN {X 0,Y 551.764,Z 932.677,A -85,B 0,C 180,E1 -3325.617,E2 -3325.617} C_VEL
LIN {X 0,Y 551.751,Z 934.957,A -85,B 0,C 180,E1 -3326.348,E2 -3326.348} C_VEL
LIN {X 0,Y 551.724,Z 936.808,A -85,B 0,C 180,E1 -3327.079,E2 -3327.079} C_VEL
LIN {X 0,Y 551.645,Z 939.186,A -85,B 0,C 180,E1 -3328.54,E2 -3328.54} C_VEL
LIN {X 0,Y 551.64,Z 940,A -85,B 0,C 180,E1 -3330,E2 -3330} C_VEL
LIN {X 0,Y 551.645,Z 939.186,A -85,B 0,C 180,E1 -3331.46,E2 -3331.46} C_VEL
LIN {X 0,Y 551.724,Z 936.81,A -85,B 0,C 180,E1 -3332.921,E2 -3332.921} C_VEL
LIN {X 0,Y 551.764,Z 933.896,A -85,B 0,C 180,E1 -3334.017,E2 -3334.017} C_VEL
LIN {X 0,Y 551.724,Z 929.949,A -85,B 0,C 180,E1 -3335.116,E2 -3335.116} C_VEL
LIN {X 0,Y 551.803,Z 924.19,A -85,B 0,C 180,E1 -3336.341,E2 -3336.341} C_VEL
LIN {X 0,Y 551.926,Z 917.238,A -85,B 0,C 180,E1 -3337.5,E2 -3337.5} C_VEL
LIN {X 0,Y 552.082,Z 908.991,A -85,B 0,C 180,E1 -3338.602,E2 -3338.602} C_VEL
LIN {X 0,Y 552.2,Z 900.539,A -85,B 0,C 180,E1 -3339.524,E2 -3339.524} C_VEL
LIN {X 0,Y 552.412,Z 890.098,A -85,B 0,C 180,E1 -3340.445,E2 -3340.445} C_VEL
LIN {X 0,Y 552.586,Z 879.311,A -85,B 0,C 180,E1 -3341.213,E2 -3341.213} C_VEL
LIN {X 0,Y 552.741,Z 868.41,A -85,B 0,C 180,E1 -3341.831,E2 -3341.831} C_VEL
LIN {X 0,Y 552.893,Z 856.764,A -85,B 0,C 180,E1 -3342.34,E2 -3342.34} C_VEL
LIN {X 0,Y 553.067,Z 843.348,A -85,B 0,C 180,E1 -3342.755,E2 -3342.755} C_VEL
LIN {X 0,Y 552.912,Z 835.493,A -85,B 0,C 180,E1 -3342.931,E2 -3342.931} C_VEL
LIN {X 0,Y 552.058,Z 830.034,A -85,B 0,C 180,E1 -3343.06,E2 -3343.06} C_VEL
LIN {X 0,Y 552.229,Z 815.361,A -85,B 0,C 180,E1 -3345.88,E2 -3345.88} C_VEL
LIN {X 0,Y 552.43,Z 801.666,A -85,B 0,C 180,E1 -3348.545,E2 -3348.545} C_VEL
LIN {X 0,Y 552.649,Z 787.971,A -85,B 0,C 180,E1 -3351.25,E2 -3351.25} C_VEL
LIN {X 0,Y 552.906,Z 774.276,A -85,B 0,C 180,E1 -3354.001,E2 -3354.001} C_VEL
LIN {X 0,Y 553.211,Z 760.581,A -85,B 0,C 180,E1 -3356.807,E2 -3356.807} C_VEL
LIN {X 0,Y 553.393,Z 744.685,A -85,B 0,C 180,E1 -3359.988,E2 -3359.988} C_VEL
LIN {X 0,Y 553.563,Z 730.564,A -85,B 0,C 180,E1 -3362.862,E2 -3362.862} C_VEL
LIN {X 0,Y 553.716,Z 717.05,A -85,B 0,C 180,E1 -3365.722,E2 -3365.722} C_VEL
LIN {X 0,Y 553.088,Z 712.294,A -85,B 0,C 180,E1 -3366.819,E2 -3366.819} C_VEL
LIN {X 0,Y 552.12,Z 707.712,A -85,B 0,C 180,E1 -3367.918,E2 -3367.918} C_VEL
LIN {X 0,Y 552.123,Z 707.708,A -85,B 0,C 180,E1 -3370.48,E2 -3370.48} C_VEL
LIN {X 0,Y 552.105,Z 707.715,A -85,B 0,C 180,E1 -3373.483,E2 -3373.483} C_VEL
LIN {X 0,Y 552.109,Z 707.707,A -85,B 0,C 180,E1 -3376.576,E2 -3376.576} C_VEL
LIN {X 0,Y 552.144,Z 707.71,A -85,B 0,C 180,E1 -3379.522,E2 -3379.522} C_VEL
LIN {X 0,Y 552.096,Z 707.708,A -85,B 0,C 180,E1 -3382.336,E2 -3382.336} C_VEL
LIN {X 0,Y 552.09,Z 707.712,A -85,B 0,C 180,E1 -3385.051,E2 -3385.051} C_VEL
LIN {X 0,Y 552.129,Z 707.712,A -85,B 0,C 180,E1 -3387.682,E2 -3387.682} C_VEL
LIN {X 0,Y 552.114,Z 707.707,A -85,B 0,C 180,E1 -3390.235,E2 -3390.235} C_VEL
LIN {X 0,Y 552.141,Z 707.704,A -85,B 0,C 180,E1 -3393,E2 -3393} C_VEL
LIN {X 0,Y 552.116,Z 707.708,A -85,B 0,C 180,E1 -3395.161,E2 -3395.161} C_VEL
LIN {X 0,Y 552.129,Z 707.706,A -85,B 0,C 180,E1 -3398.337,E2 -3398.337} C_VEL
LIN {X 0,Y 552.154,Z 707.701,A -85,B 0,C 180,E1 -3400.674,E2 -3400.674} C_VEL
LIN {X 0,Y 552.119,Z 707.713,A -85,B 0,C 180,E1 -3403.737,E2 -3403.737} C_VEL
LIN {X 0,Y 552.136,Z 707.711,A -85,B 0,C 180,E1 -3406.004,E2 -3406.004} C_VEL
LIN {X 0,Y 552.166,Z 707.699,A -85,B 0,C 180,E1 -3408.993,E2 -3408.993} C_VEL
LIN {X 0,Y 552.157,Z 707.709,A -85,B 0,C 180,E1 -3411.952,E2 -3411.952} C_VEL
LIN {X 0,Y 552.227,Z 707.692,A -85,B 0,C 180,E1 -3414.889,E2 -3414.889} C_VEL
LIN {X 0,Y 552.228,Z 707.698,A -85,B 0,C 180,E1 -3417.812,E2 -3417.812} C_VEL
LIN {X 0,Y 552.236,Z 707.693,A -85,B 0,C 180,E1 -3420.729,E2 -3420.729} C_VEL
LIN {X 0,Y 552.197,Z 707.696,A -85,B 0,C 180,E1 -3422.918,E2 -3422.918} C_VEL
LIN {X 0,Y 552.188,Z 707.701,A -85,B 0,C 180,E1 -3425.844,E2 -3425.844} C_VEL
LIN {X 0,Y 552.151,Z 707.704,A -85,B 0,C 180,E1 -3428.786,E2 -3428.786} C_VEL
LIN {X 0,Y 552.164,Z 707.702,A -85,B 0,C 180,E1 -3431.751,E2 -3431.751} C_VEL
LIN {X 0,Y 552.131,Z 707.708,A -85,B 0,C 180,E1 -3434.749,E2 -3434.749} C_VEL
LIN {X 0,Y 552.094,Z 707.71,A -85,B 0,C 180,E1 -3437.789,E2 -3437.789} C_VEL
LIN {X 0,Y 552.128,Z 707.709,A -85,B 0,C 180,E1 -3440.101,E2 -3440.101} C_VEL
LIN {X 0,Y 552.092,Z 707.717,A -85,B 0,C 180,E1 -3442.451,E2 -3442.451} C_VEL
LIN {X 0,Y 552.081,Z 707.711,A -85,B 0,C 180,E1 -3445.333,E2 -3445.333} C_VEL
LIN {X 0,Y 552.078,Z 707.713,A -85,B 0,C 180,E1 -3448.1,E2 -3448.1} C_VEL
LIN {X 0,Y 552.094,Z 707.717,A -85,B 0,C 180,E1 -3450.61,E2 -3450.61} C_VEL
LIN {X 0,Y 552.108,Z 707.71,A -85,B 0,C 180,E1 -3453.187,E2 -3453.187} C_VEL
LIN {X 0,Y 552.089,Z 707.709,A -85,B 0,C 180,E1 -3453.772,E2 -3453.772} C_VEL
LIN {X 0,Y 551.439,Z 707.796,A -85,B 0,C 180,E1 -3454.38,E2 -3454.38} C_VEL
LIN {X 0,Y 548.596,Z 708.156,A -85,B 0,C 180,E1 -3455.368,E2 -3455.368} C_VEL
LIN {X 0,Y 546.177,Z 708.46,A -85,B 0,C 180,E1 -3456.164,E2 -3456.164} C_VEL
LIN {X 0,Y 545.126,Z 708.586,A -85,B 0,C 180,E1 -3456.778,E2 -3456.778} C_VEL
LIN {X 0,Y 545.035,Z 708.595,A -85,B 0,C 180,E1 -3456.986,E2 -3456.986} C_VEL
LIN {X 0,Y 545.056,Z 708.587,A -85,B 0,C 180,E1 -3460.144,E2 -3460.144} C_VEL
LIN {X 0,Y 545.019,Z 708.597,A -85,B 0,C 180,E1 -3463.113,E2 -3463.113} C_VEL
LIN {X 0,Y 545.03,Z 708.59,A -85,B 0,C 180,E1 -3466.229,E2 -3466.229} C_VEL
LIN {X 0,Y 545.013,Z 708.599,A -85,B 0,C 180,E1 -3468.879,E2 -3468.879} C_VEL
LIN {X 0,Y 545.045,Z 708.588,A -85,B 0,C 180,E1 -3471.762,E2 -3471.762} C_VEL
LIN {X 0,Y 545.024,Z 708.592,A -85,B 0,C 180,E1 -3474.531,E2 -3474.531} C_VEL
LIN {X 0,Y 545.053,Z 708.594,A -85,B 0,C 180,E1 -3477.21,E2 -3477.21} C_VEL
LIN {X 0,Y 545.027,Z 708.591,A -85,B 0,C 180,E1 -3479.808,E2 -3479.808} C_VEL
LIN {X 0,Y 545.001,Z 708.593,A -85,B 0,C 180,E1 -3482.339,E2 -3482.339} C_VEL
LIN {X 0,Y 545.021,Z 708.593,A -85,B 0,C 180,E1 -3484.816,E2 -3484.816} C_VEL
LIN {X 0,Y 545.031,Z 708.597,A -85,B 0,C 180,E1 -3487.242,E2 -3487.242} C_VEL
LIN {X 0,Y 545.119,Z 708.578,A -85,B 0,C 180,E1 -3490.415,E2 -3490.415} C_VEL
LIN {X 0,Y 545.039,Z 708.595,A -85,B 0,C 180,E1 -3493.52,E2 -3493.52} C_VEL
LIN {X 0,Y 545.072,Z 708.588,A -85,B 0,C 180,E1 -3495.819,E2 -3495.819} C_VEL
LIN {X 0,Y 545.076,Z 708.584,A -85,B 0,C 180,E1 -3498.849,E2 -3498.849} C_VEL
LIN {X 0,Y 545.067,Z 708.589,A -85,B 0,C 180,E1 -3501.846,E2 -3501.846} C_VEL
LIN {X 0,Y 545.165,Z 708.572,A -85,B 0,C 180,E1 -3504.823,E2 -3504.823} C_VEL
LIN {X 0,Y 545.191,Z 708.576,A -85,B 0,C 180,E1 -3507.784,E2 -3507.784} C_VEL
LIN {X 0,Y 545.194,Z 708.573,A -85,B 0,C 180,E1 -3510,E2 -3510} C_VEL
LIN {X 0,Y 545.149,Z 708.574,A -85,B 0,C 180,E1 -3512.956,E2 -3512.956} C_VEL
LIN {X 0,Y 545.136,Z 708.583,A -85,B 0,C 180,E1 -3515.92,E2 -3515.92} C_VEL
LIN {X 0,Y 545.098,Z 708.58,A -85,B 0,C 180,E1 -3518.901,E2 -3518.901} C_VEL
LIN {X 0,Y 545.105,Z 708.588,A -85,B 0,C 180,E1 -3521.905,E2 -3521.905} C_VEL
LIN {X 0,Y 545.089,Z 708.581,A -85,B 0,C 180,E1 -3524.944,E2 -3524.944} C_VEL
LIN {X 0,Y 545.064,Z 708.593,A -85,B 0,C 180,E1 -3528.026,E2 -3528.026} C_VEL
LIN {X 0,Y 545.096,Z 708.585,A -85,B 0,C 180,E1 -3530.372,E2 -3530.372} C_VEL
LIN {X 0,Y 545.08,Z 708.584,A -85,B 0,C 180,E1 -3533.56,E2 -3533.56} C_VEL
LIN {X 0,Y 545.048,Z 708.594,A -85,B 0,C 180,E1 -3536.002,E2 -3536.002} C_VEL
LIN {X 0,Y 545.073,Z 708.585,A -85,B 0,C 180,E1 -3538.744,E2 -3538.744} C_VEL
LIN {X 0,Y 545.062,Z 708.586,A -85,B 0,C 180,E1 -3541.679,E2 -3541.679} C_VEL
LIN {X 0,Y 545.062,Z 708.59,A -85,B 0,C 180,E1 -3544.565,E2 -3544.565} C_VEL
LIN {X 0,Y 545.04,Z 708.587,A -85,B 0,C 180,E1 -3547.304,E2 -3547.304} C_VEL
LIN {X 0,Y 545.069,Z 708.589,A -85,B 0,C 180,E1 -3550.143,E2 -3550.143} C_VEL
LIN {X 0,Y 545.083,Z 708.582,A -85,B 0,C 180,E1 -3553.107,E2 -3553.107} C_VEL
LIN {X 0,Y 545.053,Z 708.591,A -85,B 0,C 180,E1 -3556.226,E2 -3556.226} C_VEL
LIN {X 0,Y 545.089,Z 708.588,A -85,B 0,C 180,E1 -3558.886,E2 -3558.886} C_VEL
LIN {X 0,Y 545.102,Z 708.664,A -85,B 0,C 180,E1 -3559.579,E2 -3559.579} C_VEL
LIN {X 0,Y 545.824,Z 711.578,A -85,B 0,C 180,E1 -3559.725,E2 -3559.725} C_VEL
LIN {X 0,Y 545.746,Z 721.493,A -85,B 0,C 180,E1 -3560.208,E2 -3560.208} C_VEL
LIN {X 0,Y 545.573,Z 730.784,A -85,B 0,C 180,E1 -3560.767,E2 -3560.767} C_VEL
LIN {X 0,Y 545.357,Z 739.876,A -85,B 0,C 180,E1 -3561.434,E2 -3561.434} C_VEL
LIN {X 0,Y 545.203,Z 748.925,A -85,B 0,C 180,E1 -3562.243,E2 -3562.243} C_VEL
LIN {X 0,Y 545.03,Z 756.779,A -85,B 0,C 180,E1 -3563.08,E2 -3563.08} C_VEL
LIN {X 0,Y 544.902,Z 762.699,A -85,B 0,C 180,E1 -3563.809,E2 -3563.809} C_VEL
LIN {X 0,Y 544.804,Z 769.086,A -85,B 0,C 180,E1 -3564.74,E2 -3564.74} C_VEL
LIN {X 0,Y 544.757,Z 774.353,A -85,B 0,C 180,E1 -3565.657,E2 -3565.657} C_VEL
LIN {X 0,Y 544.678,Z 779.182,A -85,B 0,C 180,E1 -3566.685,E2 -3566.685} C_VEL
LIN {X 0,Y 544.639,Z 782.754,A -85,B 0,C 180,E1 -3567.621,E2 -3567.621} C_VEL
LIN {X 0,Y 544.604,Z 786.389,A -85,B 0,C 180,E1 -3568.923,E2 -3568.923} C_VEL
LIN {X 0,Y 544.602,Z 788.23,A -85,B 0,C 180,E1 -3569.84,E2 -3569.84} C_VEL
LIN {X 0,Y 544.559,Z 789.224,A -85,B 0,C 180,E1 -3570.631,E2 -3570.631} C_VEL
LIN {X 0,Y 544.572,Z 789.799,A -85,B 0,C 180,E1 -3571.477,E2 -3571.477} C_VEL
LIN {X 0,Y 544.548,Z 789.922,A -85,B 0,C 180,E1 -3572.314,E2 -3572.314} C_VEL
LIN {X 0,Y 544.559,Z 789.558,A -85,B 0,C 180,E1 -3573.147,E2 -3573.147} C_VEL
LIN {X 0,Y 544.558,Z 787.545,A -85,B 0,C 180,E1 -3574.611,E2 -3574.611} C_VEL
LIN {X 0,Y 544.644,Z 785.303,A -85,B 0,C 180,E1 -3575.611,E2 -3575.611} C_VEL
LIN {X 0,Y 544.67,Z 781.437,A -85,B 0,C 180,E1 -3576.824,E2 -3576.824} C_VEL
LIN {X 0,Y 544.701,Z 778.261,A -85,B 0,C 180,E1 -3577.628,E2 -3577.628} C_VEL
LIN {X 0,Y 544.76,Z 772.209,A -85,B 0,C 180,E1 -3578.824,E2 -3578.824} C_VEL
LIN {X 0,Y 544.865,Z 766.076,A -85,B 0,C 180,E1 -3579.808,E2 -3579.808} C_VEL
LIN {X 0,Y 545.007,Z 760.207,A -85,B 0,C 180,E1 -3580.606,E2 -3580.606} C_VEL
LIN {X 0,Y 545.125,Z 751.543,A -85,B 0,C 180,E1 -3581.587,E2 -3581.587} C_VEL
LIN {X 0,Y 545.318,Z 743.085,A -85,B 0,C 180,E1 -3582.388,E2 -3582.388} C_VEL
LIN {X 0,Y 545.503,Z 734.695,A -85,B 0,C 180,E1 -3583.053,E2 -3583.053} C_VEL
LIN {X 0,Y 545.625,Z 725.908,A -85,B 0,C 180,E1 -3583.634,E2 -3583.634} C_VEL
LIN {X 0,Y 545.806,Z 715.947,A -85,B 0,C 180,E1 -3584.168,E2 -3584.168} C_VEL
LIN {X 0,Y 545.653,Z 711,A -85,B 0,C 180,E1 -3584.403,E2 -3584.403} C_VEL
LIN {X 0,Y 545.097,Z 708.582,A -85,B 0,C 180,E1 -3584.53,E2 -3584.53} C_VEL
LIN {X 0,Y 545.085,Z 708.589,A -85,B 0,C 180,E1 -3587.339,E2 -3587.339} C_VEL
LIN {X 0,Y 545.078,Z 708.593,A -85,B 0,C 180,E1 -3589.6,E2 -3589.6} C_VEL
LIN {X 0,Y 545.128,Z 708.583,A -85,B 0,C 180,E1 -3591.847,E2 -3591.847} C_VEL
LIN {X 0,Y 545.197,Z 708.567,A -85,B 0,C 180,E1 -3594.823,E2 -3594.823} C_VEL
LIN {X 0,Y 545.198,Z 708.577,A -85,B 0,C 180,E1 -3597.784,E2 -3597.784} C_VEL
LIN {X 0,Y 545.214,Z 708.565,A -85,B 0,C 180,E1 -3600.739,E2 -3600.739} C_VEL
LIN {X 0,Y 545.172,Z 708.569,A -85,B 0,C 180,E1 -3602.956,E2 -3602.956} C_VEL
LIN {X 0,Y 545.171,Z 708.578,A -85,B 0,C 180,E1 -3605.919,E2 -3605.919} C_VEL
LIN {X 0,Y 545.105,Z 708.577,A -85,B 0,C 180,E1 -3608.9,E2 -3608.9} C_VEL
LIN {X 0,Y 545.139,Z 708.582,A -85,B 0,C 180,E1 -3611.904,E2 -3611.904} C_VEL
LIN {X 0,Y 545.09,Z 708.579,A -85,B 0,C 180,E1 -3614.943,E2 -3614.943} C_VEL
LIN {X 0,Y 545.076,Z 708.591,A -85,B 0,C 180,E1 -3618.026,E2 -3618.026} C_VEL
LIN {X 0,Y 545.097,Z 708.586,A -85,B 0,C 180,E1 -3620.372,E2 -3620.372} C_VEL
LIN {X 0,Y 545.083,Z 708.582,A -85,B 0,C 180,E1 -3623.559,E2 -3623.559} C_VEL
LIN {X 0,Y 545.083,Z 708.587,A -85,B 0,C 180,E1 -3626,E2 -3626} C_VEL
LIN {X 0,Y 545.093,Z 708.584,A -85,B 0,C 180,E1 -3628.748,E2 -3628.748} C_VEL
LIN {X 0,Y 545.063,Z 708.585,A -85,B 0,C 180,E1 -3631.679,E2 -3631.679} C_VEL
LIN {X 0,Y 545.081,Z 708.591,A -85,B 0,C 180,E1 -3634.392,E2 -3634.392} C_VEL
LIN {X 0,Y 545.04,Z 708.589,A -85,B 0,C 180,E1 -3637.304,E2 -3637.304} C_VEL
LIN {X 0,Y 545.075,Z 708.588,A -85,B 0,C 180,E1 -3640.142,E2 -3640.142} C_VEL
LIN {X 0,Y 545.082,Z 708.586,A -85,B 0,C 180,E1 -3643.106,E2 -3643.106} C_VEL
LIN {X 0,Y 545.06,Z 708.589,A -85,B 0,C 180,E1 -3646.225,E2 -3646.225} C_VEL
LIN {X 0,Y 545.098,Z 708.59,A -85,B 0,C 180,E1 -3648.886,E2 -3648.886} C_VEL
LIN {X 0,Y 545.056,Z 708.593,A -85,B 0,C 180,E1 -3651.763,E2 -3651.763} C_VEL
LIN {X 0,Y 545.086,Z 708.797,A -85,B 0,C 180,E1 -3652.409,E2 -3652.409} C_VEL
LIN {X 0,Y 546.219,Z 714.459,A -85,B 0,C 180,E1 -3653.71,E2 -3653.71} C_VEL
LIN {X 0,Y 546.418,Z 720.774,A -85,B 0,C 180,E1 -3655.066,E2 -3655.066} C_VEL
LIN {X 0,Y 546.337,Z 733.753,A -85,B 0,C 180,E1 -3657.734,E2 -3657.734} C_VEL
LIN {X 0,Y 546.296,Z 745.678,A -85,B 0,C 180,E1 -3660.098,E2 -3660.098} C_VEL
LIN {X 0,Y 546.192,Z 762.036,A -85,B 0,C 180,E1 -3663.233,E2 -3663.233} C_VEL
LIN {X 0,Y 546.051,Z 772.319,A -85,B 0,C 180,E1 -3665.273,E2 -3665.273} C_VEL
LIN {X 0,Y 545.7,Z 786.014,A -85,B 0,C 180,E1 -3668.069,E2 -3668.069} C_VEL
LIN {X 0,Y 545.459,Z 799.709,A -85,B 0,C 180,E1 -3670.819,E2 -3670.819} C_VEL
LIN {X 0,Y 545.253,Z 813.404,A -85,B 0,C 180,E1 -3673.527,E2 -3673.527} C_VEL
LIN {X 0,Y 545.024,Z 829.055,A -85,B 0,C 180,E1 -3676.579,E2 -3676.579} C_VEL
LIN {X 0,Y 545.013,Z 830.156,A -85,B 0,C 180,E1 -3676.792,E2 -3676.792} C_VEL
LIN {X 0,Y 546.208,Z 839.362,A -85,B 0,C 180,E1 -3676.987,E2 -3676.987} C_VEL
LIN {X 0,Y 546.039,Z 851.495,A -85,B 0,C 180,E1 -3677.314,E2 -3677.314} C_VEL
LIN {X 0,Y 545.858,Z 863.511,A -85,B 0,C 180,E1 -3677.782,E2 -3677.782} C_VEL
LIN {X 0,Y 545.707,Z 875.371,A -85,B 0,C 180,E1 -3678.401,E2 -3678.401} C_VEL
LIN {X 0,Y 545.483,Z 886.481,A -85,B 0,C 180,E1 -3679.139,E2 -3679.139} C_VEL
LIN {X 0,Y 545.257,Z 896.645,A -85,B 0,C 180,E1 -3679.979,E2 -3679.979} C_VEL
LIN {X 0,Y 545.082,Z 905.785,A -85,B 0,C 180,E1 -3680.912,E2 -3680.912} C_VEL
LIN {X 0,Y 544.916,Z 914.688,A -85,B 0,C 180,E1 -3682.03,E2 -3682.03} C_VEL
LIN {X 0,Y 544.785,Z 921.848,A -85,B 0,C 180,E1 -3683.146,E2 -3683.146} C_VEL
LIN {X 0,Y 544.741,Z 928.365,A -85,B 0,C 180,E1 -3684.447,E2 -3684.447} C_VEL
LIN {X 0,Y 544.66,Z 932.677,A -85,B 0,C 180,E1 -3685.56,E2 -3685.56} C_VEL
LIN {X 0,Y 544.669,Z 934.957,A -85,B 0,C 180,E1 -3686.301,E2 -3686.301} C_VEL
LIN {X 0,Y 544.651,Z 936.808,A -85,B 0,C 180,E1 -3687.041,E2 -3687.041} C_VEL
LIN {X 0,Y 544.546,Z 939.185,A -85,B 0,C 180,E1 -3688.521,E2 -3688.521} C_VEL
LIN {X 0,Y 544.541,Z 940,A -85,B 0,C 180,E1 -3690,E2 -3690} C_VEL
LIN {X 0,Y 544.546,Z 939.186,A -85,B 0,C 180,E1 -3691.479,E2 -3691.479} C_VEL
LIN {X 0,Y 544.651,Z 936.81,A -85,B 0,C 180,E1 -3692.959,E2 -3692.959} C_VEL
LIN {X 0,Y 544.683,Z 933.896,A -85,B 0,C 180,E1 -3694.069,E2 -3694.069} C_VEL
LIN {X 0,Y 544.654,Z 929.949,A -85,B 0,C 180,E1 -3695.182,E2 -3695.182} C_VEL
LIN {X 0,Y 544.739,Z 924.704,A -85,B 0,C 180,E1 -3696.328,E2 -3696.328} C_VEL
LIN {X 0,Y 544.836,Z 918.468,A -85,B 0,C 180,E1 -3697.411,E2 -3697.411} C_VEL
LIN {X 0,Y 545.006,Z 910.478,A -85,B 0,C 180,E1 -3698.528,E2 -3698.528} C_VEL
LIN {X 0,Y 545.142,Z 902.335,A -85,B 0,C 180,E1 -3699.461,E2 -3699.461} C_VEL
LIN {X 0,Y 545.363,Z 892.401,A -85,B 0,C 180,E1 -3700.394,E2 -3700.394} C_VEL
LIN {X 0,Y 545.562,Z 882.588,A -85,B 0,C 180,E1 -3701.141,E2 -3701.141} C_VEL
LIN {X 0,Y 545.736,Z 870.176,A -85,B 0,C 180,E1 -3701.891,E2 -3701.891} C_VEL
LIN {X 0,Y 545.937,Z 857.979,A -85,B 0,C 180,E1 -3702.452,E2 -3702.452} C_VEL
LIN {X 0,Y 546.149,Z 845.176,A -85,B 0,C 180,E1 -3702.872,E2 -3702.872} C_VEL
LIN {X 0,Y 546.003,Z 836.374,A -85,B 0,C 180,E1 -3703.08,E2 -3703.08} C_VEL
LIN {X 0,Y 545.023,Z 830.034,A -85,B 0,C 180,E1 -3703.231,E2 -3703.231} C_VEL
LIN {X 0,Y 545.234,Z 815.361,A -85,B 0,C 180,E1 -3706.089,E2 -3706.089} C_VEL
LIN {X 0,Y 545.424,Z 801.666,A -85,B 0,C 180,E1 -3708.792,E2 -3708.792} C_VEL
LIN {X 0,Y 545.675,Z 787.971,A -85,B 0,C 180,E1 -3711.535,E2 -3711.535} C_VEL
LIN {X 0,Y 545.991,Z 774.276,A -85,B 0,C 180,E1 -3714.325,E2 -3714.325} C_VEL
LIN {X 0,Y 546.217,Z 762.243,A -85,B 0,C 180,E1 -3716.765,E2 -3716.765} C_VEL
LIN {X 0,Y 546.425,Z 746.696,A -85,B 0,C 180,E1 -3719.894,E2 -3719.894} C_VEL
LIN {X 0,Y 546.616,Z 733.091,A -85,B 0,C 180,E1 -3722.684,E2 -3722.684} C_VEL
LIN {X 0,Y 546.772,Z 720.682,A -85,B 0,C 180,E1 -3725.339,E2 -3725.339} C_VEL
LIN {X 0,Y 546.726,Z 716.592,A -85,B 0,C 180,E1 -3726.251,E2 -3726.251} C_VEL
LIN {X 0,Y 545.052,Z 708.593,A -85,B 0,C 180,E1 -3728.197,E2 -3728.197} C_VEL
LIN {X 0,Y 545.093,Z 708.585,A -85,B 0,C 180,E1 -3730.474,E2 -3730.474} C_VEL
LIN {X 0,Y 545.083,Z 708.59,A -85,B 0,C 180,E1 -3733.106,E2 -3733.106} C_VEL
LIN {X 0,Y 545.07,Z 708.584,A -85,B 0,C 180,E1 -3736.224,E2 -3736.224} C_VEL
LIN {X 0,Y 545.098,Z 708.583,A -85,B 0,C 180,E1 -3738.887,E2 -3738.887} C_VEL
LIN {X 0,Y 545.056,Z 708.59,A -85,B 0,C 180,E1 -3741.763,E2 -3741.763} C_VEL
LIN {X 0,Y 545.041,Z 708.587,A -85,B 0,C 180,E1 -3744.532,E2 -3744.532} C_VEL
LIN {X 0,Y 545.085,Z 708.586,A -85,B 0,C 180,E1 -3747.213,E2 -3747.213} C_VEL
LIN {X 0,Y 545.067,Z 708.59,A -85,B 0,C 180,E1 -3749.811,E2 -3749.811} C_VEL
LIN {X 0,Y 545.084,Z 708.582,A -85,B 0,C 180,E1 -3752.344,E2 -3752.344} C_VEL
LIN {X 0,Y 545.12,Z 708.577,A -85,B 0,C 180,E1 -3754.821,E2 -3754.821} C_VEL
LIN {X 0,Y 545.039,Z 708.59,A -85,B 0,C 180,E1 -3757.242,E2 -3757.242} C_VEL
LIN {X 0,Y 545.12,Z 708.579,A -85,B 0,C 180,E1 -3760.415,E2 -3760.415} C_VEL
LIN {X 0,Y 545.075,Z 708.588,A -85,B 0,C 180,E1 -3763.521,E2 -3763.521} C_VEL
LIN {X 0,Y 545.097,Z 708.588,A -85,B 0,C 180,E1 -3765.82,E2 -3765.82} C_VEL
LIN {X 0,Y 545.121,Z 708.577,A -85,B 0,C 180,E1 -3768.849,E2 -3768.849} C_VEL
LIN {X 0,Y 545.128,Z 708.584,A -85,B 0,C 180,E1 -3771.847,E2 -3771.847} C_VEL
LIN {X 0,Y 545.203,Z 708.568,A -85,B 0,C 180,E1 -3774.823,E2 -3774.823} C_VEL
LIN {X 0,Y 545.199,Z 708.573,A -85,B 0,C 180,E1 -3777.784,E2 -3777.784} C_VEL
LIN {X 0,Y 545.207,Z 708.568,A -85,B 0,C 180,E1 -3780.739,E2 -3780.739} C_VEL
LIN {X 0,Y 545.164,Z 708.572,A -85,B 0,C 180,E1 -3782.956,E2 -3782.956} C_VEL
LIN {X 0,Y 545.16,Z 708.578,A -85,B 0,C 180,E1 -3785.92,E2 -3785.92} C_VEL
LIN {X 0,Y 545.108,Z 708.581,A -85,B 0,C 180,E1 -3788.9,E2 -3788.9} C_VEL
LIN {X 0,Y 545.107,Z 708.583,A -85,B 0,C 180,E1 -3791.905,E2 -3791.905} C_VEL
LIN {X 0,Y 545.084,Z 708.584,A -85,B 0,C 180,E1 -3794.944,E2 -3794.944} C_VEL
LIN {X 0,Y 545.061,Z 708.589,A -85,B 0,C 180,E1 -3798.027,E2 -3798.027} C_VEL
LIN {X 0,Y 545.094,Z 708.588,A -85,B 0,C 180,E1 -3800.372,E2 -3800.372} C_VEL
LIN {X 0,Y 545.076,Z 708.583,A -85,B 0,C 180,E1 -3803.56,E2 -3803.56} C_VEL
LIN {X 0,Y 545.038,Z 708.59,A -85,B 0,C 180,E1 -3806.003,E2 -3806.003} C_VEL
LIN {X 0,Y 545.066,Z 708.593,A -85,B 0,C 180,E1 -3808.743,E2 -3808.743} C_VEL
LIN {X 0,Y 545.061,Z 708.585,A -85,B 0,C 180,E1 -3811.679,E2 -3811.679} C_VEL
LIN {X 0,Y 545.05,Z 708.594,A -85,B 0,C 180,E1 -3814.566,E2 -3814.566} C_VEL
LIN {X 0,Y 545.035,Z 708.595,A -85,B 0,C 180,E1 -3816.986,E2 -3816.986} C_VEL
LIN {X 0,Y 544.353,Z 708.676,A -85,B 0,C 180,E1 -3817.603,E2 -3817.603} C_VEL
LIN {X 0,Y 541.495,Z 709.036,A -85,B 0,C 180,E1 -3818.604,E2 -3818.604} C_VEL
LIN {X 0,Y 539.093,Z 709.331,A -85,B 0,C 180,E1 -3819.41,E2 -3819.41} C_VEL
LIN {X 0,Y 538.066,Z 709.457,A -85,B 0,C 180,E1 -3820.032,E2 -3820.032} C_VEL
LIN {X 0,Y 537.984,Z 709.468,A -85,B 0,C 180,E1 -3820.242,E2 -3820.242} C_VEL
LIN {X 0,Y 537.972,Z 709.476,A -85,B 0,C 180,E1 -3822.981,E2 -3822.981} C_VEL
LIN {X 0,Y 538.003,Z 709.464,A -85,B 0,C 180,E1 -3825.929,E2 -3825.929} C_VEL
LIN {X 0,Y 537.995,Z 709.471,A -85,B 0,C 180,E1 -3829.26,E2 -3829.26} C_VEL
LIN {X 0,Y 537.983,Z 709.467,A -85,B 0,C 180,E1 -3832.121,E2 -3832.121} C_VEL
LIN {X 0,Y 537.994,Z 709.471,A -85,B 0,C 180,E1 -3835.386,E2 -3835.386} C_VEL
LIN {X 0,Y 537.997,Z 709.465,A -85,B 0,C 180,E1 -3838.116,E2 -3838.116} C_VEL
LIN {X 0,Y 537.986,Z 709.474,A -85,B 0,C 180,E1 -3841.095,E2 -3841.095} C_VEL
LIN {X 0,Y 537.97,Z 709.472,A -85,B 0,C 180,E1 -3843.629,E2 -3843.629} C_VEL
LIN {X 0,Y 538.009,Z 709.464,A -85,B 0,C 180,E1 -3846.123,E2 -3846.123} C_VEL
LIN {X 0,Y 538.036,Z 709.468,A -85,B 0,C 180,E1 -3849.348,E2 -3849.348} C_VEL
LIN {X 0,Y 538.007,Z 709.468,A -85,B 0,C 180,E1 -3851.729,E2 -3851.729} C_VEL
LIN {X 0,Y 538.041,Z 709.462,A -85,B 0,C 180,E1 -3854.856,E2 -3854.856} C_VEL
LIN {X 0,Y 538.04,Z 709.463,A -85,B 0,C 180,E1 -3857.937,E2 -3857.937} C_VEL
LIN {X 0,Y 538.026,Z 709.463,A -85,B 0,C 180,E1 -3860.982,E2 -3860.982} C_VEL
LIN {X 0,Y 538.083,Z 709.458,A -85,B 0,C 180,E1 -3864.002,E2 -3864.002} C_VEL
LIN {X 0,Y 538.116,Z 709.452,A -85,B 0,C 180,E1 -3867.005,E2 -3867.005} C_VEL
LIN {X 0,Y 538.162,Z 709.449,A -85,B 0,C 180,E1 -3870,E2 -3870} C_VEL
LIN {X 0,Y 538.117,Z 709.451,A -85,B 0,C 180,E1 -3872.995,E2 -3872.995} C_VEL
LIN {X 0,Y 538.092,Z 709.459,A -85,B 0,C 180,E1 -3875.998,E2 -3875.998} C_VEL
LIN {X 0,Y 538.051,Z 709.458,A -85,B 0,C 180,E1 -3879.018,E2 -3879.018} C_VEL
LIN {X 0,Y 538.065,Z 709.463,A -85,B 0,C 180,E1 -3882.063,E2 -3882.063} C_VEL
LIN {X 0,Y 538.048,Z 709.459,A -85,B 0,C 180,E1 -3885.144,E2 -3885.144} C_VEL
LIN {X 0,Y 538.017,Z 709.468,A -85,B 0,C 180,E1 -3888.271,E2 -3888.271} C_VEL
LIN {X 0,Y 538.041,Z 709.461,A -85,B 0,C 180,E1 -3890.651,E2 -3890.651} C_VEL
LIN {X 0,Y 538.011,Z 709.469,A -85,B 0,C 180,E1 -3893.878,E2 -3893.878} C_VEL
LIN {X 0,Y 538.012,Z 709.469,A -85,B 0,C 180,E1 -3896.368,E2 -3896.368} C_VEL
LIN {X 0,Y 538.034,Z 709.46,A -85,B 0,C 180,E1 -3898.933,E2 -3898.933} C_VEL
LIN {X 0,Y 538.014,Z 709.466,A -85,B 0,C 180,E1 -3901.887,E2 -3901.887} C_VEL
LIN {X 0,Y 538.012,Z 709.467,A -85,B 0,C 180,E1 -3904.617,E2 -3904.617} C_VEL
LIN {X 0,Y 538.008,Z 709.463,A -85,B 0,C 180,E1 -3907.17,E2 -3907.17} C_VEL
LIN {X 0,Y 538.026,Z 709.462,A -85,B 0,C 180,E1 -3909.797,E2 -3909.797} C_VEL
LIN {X 0,Y 538.023,Z 709.465,A -85,B 0,C 180,E1 -3912.786,E2 -3912.786} C_VEL
LIN {X 0,Y 538.022,Z 709.463,A -85,B 0,C 180,E1 -3915.927,E2 -3915.927} C_VEL
LIN {X 0,Y 538.069,Z 709.46,A -85,B 0,C 180,E1 -3919.226,E2 -3919.226} C_VEL
LIN {X 0,Y 538.057,Z 709.478,A -85,B 0,C 180,E1 -3919.414,E2 -3919.414} C_VEL
LIN {X 0,Y 539.011,Z 713.622,A -85,B 0,C 180,E1 -3919.624,E2 -3919.624} C_VEL
LIN {X 0,Y 538.854,Z 724.053,A -85,B 0,C 180,E1 -3920.155,E2 -3920.155} C_VEL
LIN {X 0,Y 538.625,Z 733.345,A -85,B 0,C 180,E1 -3920.74,E2 -3920.74} C_VEL
LIN {X 0,Y 538.401,Z 742.272,A -85,B 0,C 180,E1 -3921.424,E2 -3921.424} C_VEL
LIN {X 0,Y 538.268,Z 750.122,A -85,B 0,C 180,E1 -3922.145,E2 -3922.145} C_VEL
LIN {X 0,Y 538.074,Z 758.534,A -85,B 0,C 180,E1 -3923.071,E2 -3923.071} C_VEL
LIN {X 0,Y 537.914,Z 763.87,A -85,B 0,C 180,E1 -3923.757,E2 -3923.757} C_VEL
LIN {X 0,Y 537.804,Z 770.069,A -85,B 0,C 180,E1 -3924.701,E2 -3924.701} C_VEL
LIN {X 0,Y 537.681,Z 775.975,A -85,B 0,C 180,E1 -3925.802,E2 -3925.802} C_VEL
LIN {X 0,Y 537.594,Z 780.281,A -85,B 0,C 180,E1 -3926.791,E2 -3926.791} C_VEL
LIN {X 0,Y 537.581,Z 783.179,A -85,B 0,C 180,E1 -3927.587,E2 -3927.587} C_VEL
LIN {X 0,Y 537.544,Z 785.682,A -85,B 0,C 180,E1 -3928.468,E2 -3928.468} C_VEL
LIN {X 0,Y 537.515,Z 788.169,A -85,B 0,C 180,E1 -3929.65,E2 -3929.65} C_VEL
LIN {X 0,Y 537.475,Z 789.843,A -85,B 0,C 180,E1 -3931.175,E2 -3931.175} C_VEL
LIN {X 0,Y 537.451,Z 790.139,A -85,B 0,C 180,E1 -3931.916,E2 -3931.916} C_VEL
LIN {X 0,Y 537.464,Z 789.904,A -85,B 0,C 180,E1 -3932.771,E2 -3932.771} C_VEL
LIN {X 0,Y 537.454,Z 789.263,A -85,B 0,C 180,E1 -3933.602,E2 -3933.602} C_VEL
LIN {X 0,Y 537.464,Z 788.16,A -85,B 0,C 180,E1 -3934.457,E2 -3934.457} C_VEL
LIN {X 0,Y 537.555,Z 785.547,A -85,B 0,C 180,E1 -3935.68,E2 -3935.68} C_VEL
LIN {X 0,Y 537.594,Z 781.78,A -85,B 0,C 180,E1 -3936.909,E2 -3936.909} C_VEL
LIN {X 0,Y 537.67,Z 778.667,A -85,B 0,C 180,E1 -3937.724,E2 -3937.724} C_VEL
LIN {X 0,Y 537.758,Z 772.743,A -85,B 0,C 180,E1 -3938.936,E2 -3938.936} C_VEL
LIN {X 0,Y 537.883,Z 766.678,A -85,B 0,C 180,E1 -3939.941,E2 -3939.941} C_VEL
LIN {X 0,Y 538.071,Z 760.936,A -85,B 0,C 180,E1 -3940.743,E2 -3940.743} C_VEL
LIN {X 0,Y 538.211,Z 752.352,A -85,B 0,C 180,E1 -3941.736,E2 -3941.736} C_VEL
LIN {X 0,Y 538.413,Z 744.061,A -85,B 0,C 180,E1 -3942.529,E2 -3942.529} C_VEL
LIN {X 0,Y 538.628,Z 735.376,A -85,B 0,C 180,E1 -3943.221,E2 -3943.221} C_VEL
LIN {X 0,Y 538.754,Z 726.51,A -85,B 0,C 180,E1 -3943.809,E2 -3943.809} C_VEL
LIN {X 0,Y 538.946,Z 716.432,A -85,B 0,C 180,E1 -3944.349,E2 -3944.349} C_VEL
LIN {X 0,Y 538.939,Z 713.36,A -85,B 0,C 180,E1 -3944.494,E2 -3944.494} C_VEL
LIN {X 0,Y 538.037,Z 709.463,A -85,B 0,C 180,E1 -3944.71,E2 -3944.71} C_VEL
LIN {X 0,Y 538.068,Z 709.463,A -85,B 0,C 180,E1 -3947.937,E2 -3947.937} C_VEL
LIN {X 0,Y 538.061,Z 709.459,A -85,B 0,C 180,E1 -3950.982,E2 -3950.982} C_VEL
LIN {X 0,Y 538.095,Z 709.457,A -85,B 0,C 180,E1 -3954.002,E2 -3954.002} C_VEL
LIN {X 0,Y 538.134,Z 709.449,A -85,B 0,C 180,E1 -3957.005,E2 -3957.005} C_VEL
LIN {X 0,Y 538.179,Z 709.449,A -85,B 0,C 180,E1 -3960,E2 -3960} C_VEL
LIN {X 0,Y 538.138,Z 709.445,A -85,B 0,C 180,E1 -3962.994,E2 -3962.994} C_VEL
LIN {X 0,Y 538.125,Z 709.456,A -85,B 0,C 180,E1 -3965.997,E2 -3965.997} C_VEL
LIN {X 0,Y 538.058,Z 709.455,A -85,B 0,C 180,E1 -3969.018,E2 -3969.018} C_VEL
LIN {X 0,Y 538.087,Z 709.46,A -85,B 0,C 180,E1 -3972.062,E2 -3972.062} C_VEL
LIN {X 0,Y 538.05,Z 709.456,A -85,B 0,C 180,E1 -3975.144,E2 -3975.144} C_VEL
LIN {X 0,Y 538.03,Z 709.468,A -85,B 0,C 180,E1 -3978.27,E2 -3978.27} C_VEL
LIN {X 0,Y 538.042,Z 709.46,A -85,B 0,C 180,E1 -3980.651,E2 -3980.651} C_VEL
LIN {X 0,Y 538.006,Z 709.467,A -85,B 0,C 180,E1 -3983.888,E2 -3983.888} C_VEL
LIN {X 0,Y 538.045,Z 709.466,A -85,B 0,C 180,E1 -3986.367,E2 -3986.367} C_VEL
LIN {X 0,Y 538.035,Z 709.461,A -85,B 0,C 180,E1 -3988.933,E2 -3988.933} C_VEL
LIN {X 0,Y 538.018,Z 709.464,A -85,B 0,C 180,E1 -3991.888,E2 -3991.888} C_VEL
LIN {X 0,Y 538.018,Z 709.47,A -85,B 0,C 180,E1 -3994.618,E2 -3994.618} C_VEL
LIN {X 0,Y 538.008,Z 709.466,A -85,B 0,C 180,E1 -3997.17,E2 -3997.17} C_VEL
LIN {X 0,Y 538.031,Z 709.463,A -85,B 0,C 180,E1 -3999.796,E2 -3999.796} C_VEL
LIN {X 0,Y 538.022,Z 709.47,A -85,B 0,C 180,E1 -4002.786,E2 -4002.786} C_VEL
LIN {X 0,Y 538.036,Z 709.464,A -85,B 0,C 180,E1 -4005.14,E2 -4005.14} C_VEL
LIN {X 0,Y 538.044,Z 709.465,A -85,B 0,C 180,E1 -4008.228,E2 -4008.228} C_VEL
LIN {X 0,Y 538.017,Z 709.472,A -85,B 0,C 180,E1 -4011.17,E2 -4011.17} C_VEL
LIN {X 0,Y 538.025,Z 709.578,A -85,B 0,C 180,E1 -4012.168,E2 -4012.168} C_VEL
LIN {X 0,Y 539.397,Z 716.923,A -85,B 0,C 180,E1 -4013.884,E2 -4013.884} C_VEL
LIN {X 0,Y 539.428,Z 726.432,A -85,B 0,C 180,E1 -4015.928,E2 -4015.928} C_VEL
LIN {X 0,Y 539.348,Z 740.313,A -85,B 0,C 180,E1 -4018.791,E2 -4018.791} C_VEL
LIN {X 0,Y 539.193,Z 755.656,A -85,B 0,C 180,E1 -4021.804,E2 -4021.804} C_VEL
LIN {X 0,Y 539.069,Z 769.636,A -85,B 0,C 180,E1 -4024.518,E2 -4024.518} C_VEL
LIN {X 0,Y 538.955,Z 778.187,A -85,B 0,C 180,E1 -4026.156,E2 -4026.156} C_VEL
LIN {X 0,Y 538.665,Z 791.883,A -85,B 0,C 180,E1 -4028.974,E2 -4028.974} C_VEL
LIN {X 0,Y 538.357,Z 807.426,A -85,B 0,C 180,E1 -4032.113,E2 -4032.113} C_VEL
LIN {X 0,Y 538.1,Z 822.594,A -85,B 0,C 180,E1 -4035.128,E2 -4035.128} C_VEL
LIN {X 0,Y 537.975,Z 830.156,A -85,B 0,C 180,E1 -4036.616,E2 -4036.616} C_VEL
LIN {X 0,Y 539.3,Z 839.361,A -85,B 0,C 180,E1 -4036.817,E2 -4036.817} C_VEL
LIN {X 0,Y 539.127,Z 851.495,A -85,B 0,C 180,E1 -4037.148,E2 -4037.148} C_VEL
LIN {X 0,Y 538.931,Z 863.51,A -85,B 0,C 180,E1 -4037.622,E2 -4037.622} C_VEL
LIN {X 0,Y 538.757,Z 875.148,A -85,B 0,C 180,E1 -4038.236,E2 -4038.236} C_VEL
LIN {X 0,Y 538.501,Z 886.482,A -85,B 0,C 180,E1 -4038.996,E2 -4038.996} C_VEL
LIN {X 0,Y 538.223,Z 896.645,A -85,B 0,C 180,E1 -4039.847,E2 -4039.847} C_VEL
LIN {X 0,Y 538.055,Z 905.785,A -85,B 0,C 180,E1 -4040.793,E2 -4040.793} C_VEL
LIN {X 0,Y 537.851,Z 914.688,A -85,B 0,C 180,E1 -4041.925,E2 -4041.925} C_VEL
LIN {X 0,Y 537.729,Z 921.848,A -85,B 0,C 180,E1 -4043.056,E2 -4043.056} C_VEL
LIN {X 0,Y 537.676,Z 928.365,A -85,B 0,C 180,E1 -4044.374,E2 -4044.374} C_VEL
LIN {X 0,Y 537.558,Z 932.677,A -85,B 0,C 180,E1 -4045.501,E2 -4045.501} C_VEL
LIN {X 0,Y 537.591,Z 934.958,A -85,B 0,C 180,E1 -4046.252,E2 -4046.252} C_VEL
LIN {X 0,Y 537.551,Z 936.807,A -85,B 0,C 180,E1 -4047.002,E2 -4047.002} C_VEL
LIN {X 0,Y 537.489,Z 938.196,A -85,B 0,C 180,E1 -4047.752,E2 -4047.752} C_VEL
LIN {X 0,Y 537.442,Z 939.785,A -85,B 0,C 180,E1 -4049.251,E2 -4049.251} C_VEL
LIN {X 0,Y 537.442,Z 940,A -85,B 0,C 180,E1 -4050,E2 -4050} C_VEL
LIN {X 0,Y 537.451,Z 939.185,A -85,B 0,C 180,E1 -4051.499,E2 -4051.499} C_VEL
LIN {X 0,Y 537.489,Z 938.198,A -85,B 0,C 180,E1 -4052.248,E2 -4052.248} C_VEL
LIN {X 0,Y 537.551,Z 936.81,A -85,B 0,C 180,E1 -4052.998,E2 -4052.998} C_VEL
LIN {X 0,Y 537.603,Z 933.896,A -85,B 0,C 180,E1 -4054.123,E2 -4054.123} C_VEL
LIN {X 0,Y 537.587,Z 929.949,A -85,B 0,C 180,E1 -4055.251,E2 -4055.251} C_VEL
LIN {X 0,Y 537.65,Z 925.08,A -85,B 0,C 180,E1 -4056.335,E2 -4056.335} C_VEL
LIN {X 0,Y 537.791,Z 918.468,A -85,B 0,C 180,E1 -4057.509,E2 -4057.509} C_VEL
LIN {X 0,Y 537.972,Z 910.478,A -85,B 0,C 180,E1 -4058.64,E2 -4058.64} C_VEL
LIN {X 0,Y 538.118,Z 902.335,A -85,B 0,C 180,E1 -4059.585,E2 -4059.585} C_VEL
LIN {X 0,Y 538.353,Z 892.4,A -85,B 0,C 180,E1 -4060.531,E2 -4060.531} C_VEL
LIN {X 0,Y 538.593,Z 882.589,A -85,B 0,C 180,E1 -4061.287,E2 -4061.287} C_VEL
LIN {X 0,Y 538.752,Z 871.513,A -85,B 0,C 180,E1 -4061.975,E2 -4061.975} C_VEL
LIN {X 0,Y 538.99,Z 859.107,A -85,B 0,C 180,E1 -4062.568,E2 -4062.568} C_VEL
LIN {X 0,Y 539.223,Z 846.089,A -85,B 0,C 180,E1 -4063.017,E2 -4063.017} C_VEL
LIN {X 0,Y 539.158,Z 837.657,A -85,B 0,C 180,E1 -4063.222,E2 -4063.222} C_VEL
LIN {X 0,Y 537.97,Z 830.034,A -85,B 0,C 180,E1 -4063.408,E2 -4063.408} C_VEL
LIN {X 0,Y 538.22,Z 815.361,A -85,B 0,C 180,E1 -4066.305,E2 -4066.305} C_VEL
LIN {X 0,Y 538.432,Z 801.666,A -85,B 0,C 180,E1 -4069.045,E2 -4069.045} C_VEL
LIN {X 0,Y 538.721,Z 788.146,A -85,B 0,C 180,E1 -4071.791,E2 -4071.791} C_VEL
LIN {X 0,Y 539.013,Z 775.738,A -85,B 0,C 180,E1 -4074.334,E2 -4074.334} C_VEL
LIN {X 0,Y 539.219,Z 761.603,A -85,B 0,C 180,E1 -4077.141,E2 -4077.141} C_VEL
LIN {X 0,Y 539.476,Z 746.038,A -85,B 0,C 180,E1 -4080.319,E2 -4080.319} C_VEL
LIN {X 0,Y 539.701,Z 732.506,A -85,B 0,C 180,E1 -4083.156,E2 -4083.156} C_VEL
LIN {X 0,Y 539.918,Z 720.201,A -85,B 0,C 180,E1 -4085.856,E2 -4085.856} C_VEL
LIN {X 0,Y 539.411,Z 716.115,A -85,B 0,C 180,E1 -4086.822,E2 -4086.822} C_VEL
LIN {X 0,Y 538.008,Z 709.471,A -85,B 0,C 180,E1 -4088.485,E2 -4088.485} C_VEL
LIN {X 0,Y 538.054,Z 709.464,A -85,B 0,C 180,E1 -4090.775,E2 -4090.775} C_VEL
LIN {X 0,Y 538.027,Z 709.462,A -85,B 0,C 180,E1 -4094.074,E2 -4094.074} C_VEL
LIN {X 0,Y 538.028,Z 709.465,A -85,B 0,C 180,E1 -4097.013,E2 -4097.013} C_VEL
LIN {X 0,Y 538.057,Z 709.465,A -85,B 0,C 180,E1 -4099.252,E2 -4099.252} C_VEL
LIN {X 0,Y 537.996,Z 709.465,A -85,B 0,C 180,E1 -4102.122,E2 -4102.122} C_VEL
LIN {X 0,Y 538.003,Z 709.465,A -85,B 0,C 180,E1 -4104.916,E2 -4104.916} C_VEL
LIN {X 0,Y 538.029,Z 709.469,A -85,B 0,C 180,E1 -4107.618,E2 -4107.618} C_VEL
LIN {X 0,Y 538.02,Z 709.463,A -85,B 0,C 180,E1 -4110.239,E2 -4110.239} C_VEL
LIN {X 0,Y 538.06,Z 709.457,A -85,B 0,C 180,E1 -4112.796,E2 -4112.796} C_VEL
LIN {X 0,Y 538.03,Z 709.464,A -85,B 0,C 180,E1 -4115.292,E2 -4115.292} C_VEL
LIN {X 0,Y 538.018,Z 709.467,A -85,B 0,C 180,E1 -4118.042,E2 -4118.042} C_VEL
LIN {X 0,Y 538.036,Z 709.46,A -85,B 0,C 180,E1 -4120.94,E2 -4120.94} C_VEL
LIN {X 0,Y 538.022,Z 709.464,A -85,B 0,C 180,E1 -4123.299,E2 -4123.299} C_VEL
LIN {X 0,Y 538.066,Z 709.462,A -85,B 0,C 180,E1 -4125.631,E2 -4125.631} C_VEL
LIN {X 0,Y 538.081,Z 709.455,A -85,B 0,C 180,E1 -4128.702,E2 -4128.702} C_VEL
LIN {X 0,Y 538.085,Z 709.46,A -85,B 0,C 180,E1 -4131.74,E2 -4131.74} C_VEL
LIN {X 0,Y 538.122,Z 709.457,A -85,B 0,C 180,E1 -4134.003,E2 -4134.003} C_VEL
LIN {X 0,Y 538.129,Z 709.448,A -85,B 0,C 180,E1 -4137.006,E2 -4137.006} C_VEL
LIN {X 0,Y 538.178,Z 709.449,A -85,B 0,C 180,E1 -4140,E2 -4140} C_VEL
LIN {X 0,Y 538.132,Z 709.448,A -85,B 0,C 180,E1 -4142.995,E2 -4142.995} C_VEL
LIN {X 0,Y 538.112,Z 709.457,A -85,B 0,C 180,E1 -4145.998,E2 -4145.998} C_VEL
LIN {X 0,Y 538.059,Z 709.458,A -85,B 0,C 180,E1 -4149.018,E2 -4149.018} C_VEL
LIN {X 0,Y 538.066,Z 709.462,A -85,B 0,C 180,E1 -4152.063,E2 -4152.063} C_VEL
LIN {X 0,Y 538.044,Z 709.46,A -85,B 0,C 180,E1 -4155.144,E2 -4155.144} C_VEL
LIN {X 0,Y 538.014,Z 709.47,A -85,B 0,C 180,E1 -4158.271,E2 -4158.271} C_VEL
LIN {X 0,Y 538.04,Z 709.467,A -85,B 0,C 180,E1 -4160.652,E2 -4160.652} C_VEL
LIN {X 0,Y 538.009,Z 709.465,A -85,B 0,C 180,E1 -4163.878,E2 -4163.878} C_VEL
LIN {X 0,Y 537.983,Z 709.473,A -85,B 0,C 180,E1 -4166.37,E2 -4166.37} C_VEL
LIN {X 0,Y 538.033,Z 709.466,A -85,B 0,C 180,E1 -4168.933,E2 -4168.933} C_VEL
LIN {X 0,Y 538.012,Z 709.464,A -85,B 0,C 180,E1 -4171.887,E2 -4171.887} C_VEL
LIN {X 0,Y 538,Z 709.472,A -85,B 0,C 180,E1 -4174.615,E2 -4174.615} C_VEL
LIN {X 0,Y 537.987,Z 709.47,A -85,B 0,C 180,E1 -4177.167,E2 -4177.167} C_VEL
LIN {X 0,Y 538.002,Z 709.465,A -85,B 0,C 180,E1 -4179.799,E2 -4179.799} C_VEL
LIN {X 0,Y 537.984,Z 709.468,A -85,B 0,C 180,E1 -4180.242,E2 -4180.242} C_VEL
LIN {X 0,Y 537.322,Z 709.557,A -85,B 0,C 180,E1 -4180.867,E2 -4180.867} C_VEL
LIN {X 0,Y 534.468,Z 709.913,A -85,B 0,C 180,E1 -4181.882,E2 -4181.882} C_VEL
LIN {X 0,Y 532.051,Z 710.213,A -85,B 0,C 180,E1 -4182.699,E2 -4182.699} C_VEL
LIN {X 0,Y 531.012,Z 710.339,A -85,B 0,C 180,E1 -4183.33,E2 -4183.33} C_VEL
LIN {X 0,Y 530.927,Z 710.347,A -85,B 0,C 180,E1 -4183.543,E2 -4183.543} C_VEL
LIN {X 0,Y 530.928,Z 710.349,A -85,B 0,C 180,E1 -4186.501,E2 -4186.501} C_VEL
LIN {X 0,Y 530.942,Z 710.346,A -85,B 0,C 180,E1 -4189.563,E2 -4189.563} C_VEL
LIN {X 0,Y 530.934,Z 710.347,A -85,B 0,C 180,E1 -4192.49,E2 -4192.49} C_VEL
LIN {X 0,Y 530.967,Z 710.348,A -85,B 0,C 180,E1 -4195.308,E2 -4195.308} C_VEL
LIN {X 0,Y 530.955,Z 710.343,A -85,B 0,C 180,E1 -4198.031,E2 -4198.031} C_VEL
LIN {X 0,Y 530.964,Z 710.347,A -85,B 0,C 180,E1 -4200.88,E2 -4200.88} C_VEL
LIN {X 0,Y 530.94,Z 710.351,A -85,B 0,C 180,E1 -4203.253,E2 -4203.253} C_VEL
LIN {X 0,Y 530.954,Z 710.344,A -85,B 0,C 180,E1 -4205.969,E2 -4205.969} C_VEL
LIN {X 0,Y 530.998,Z 710.343,A -85,B 0,C 180,E1 -4209.062,E2 -4209.062} C_VEL
LIN {X 0,Y 530.97,Z 710.347,A -85,B 0,C 180,E1 -4211.478,E2 -4211.478} C_VEL
LIN {X 0,Y 530.986,Z 710.339,A -85,B 0,C 180,E1 -4214.65,E2 -4214.65} C_VEL
LIN {X 0,Y 531.011,Z 710.341,A -85,B 0,C 180,E1 -4217.774,E2 -4217.774} C_VEL
LIN {X 0,Y 530.991,Z 710.339,A -85,B 0,C 180,E1 -4220.861,E2 -4220.861} C_VEL
LIN {X 0,Y 531.043,Z 710.336,A -85,B 0,C 180,E1 -4223.922,E2 -4223.922} C_VEL
LIN {X 0,Y 531.057,Z 710.331,A -85,B 0,C 180,E1 -4226.966,E2 -4226.966} C_VEL
LIN {X 0,Y 531.131,Z 710.325,A -85,B 0,C 180,E1 -4230,E2 -4230} C_VEL
LIN {X 0,Y 531.059,Z 710.33,A -85,B 0,C 180,E1 -4233.035,E2 -4233.035} C_VEL
LIN {X 0,Y 531.051,Z 710.336,A -85,B 0,C 180,E1 -4236.078,E2 -4236.078} C_VEL
LIN {X 0,Y 531.014,Z 710.336,A -85,B 0,C 180,E1 -4239.139,E2 -4239.139} C_VEL
LIN {X 0,Y 531.054,Z 710.336,A -85,B 0,C 180,E1 -4241.671,E2 -4241.671} C_VEL
LIN {X 0,Y 531.036,Z 710.332,A -85,B 0,C 180,E1 -4244.956,E2 -4244.956} C_VEL
LIN {X 0,Y 530.984,Z 710.344,A -85,B 0,C 180,E1 -4247.724,E2 -4247.724} C_VEL
LIN {X 0,Y 531.029,Z 710.34,A -85,B 0,C 180,E1 -4250.127,E2 -4250.127} C_VEL
LIN {X 0,Y 530.948,Z 710.345,A -85,B 0,C 180,E1 -4252.573,E2 -4252.573} C_VEL
LIN {X 0,Y 530.961,Z 710.341,A -85,B 0,C 180,E1 -4255.06,E2 -4255.06} C_VEL
LIN {X 0,Y 530.969,Z 710.342,A -85,B 0,C 180,E1 -4257.598,E2 -4257.598} C_VEL
LIN {X 0,Y 530.965,Z 710.35,A -85,B 0,C 180,E1 -4260.198,E2 -4260.198} C_VEL
LIN {X 0,Y 530.97,Z 710.341,A -85,B 0,C 180,E1 -4262.867,E2 -4262.867} C_VEL
LIN {X 0,Y 530.958,Z 710.342,A -85,B 0,C 180,E1 -4265.62,E2 -4265.62} C_VEL
LIN {X 0,Y 530.97,Z 710.345,A -85,B 0,C 180,E1 -4268.653,E2 -4268.653} C_VEL
LIN {X 0,Y 530.997,Z 710.336,A -85,B 0,C 180,E1 -4271.436,E2 -4271.436} C_VEL
LIN {X 0,Y 530.977,Z 710.347,A -85,B 0,C 180,E1 -4274.548,E2 -4274.548} C_VEL
LIN {X 0,Y 530.986,Z 710.341,A -85,B 0,C 180,E1 -4277.834,E2 -4277.834} C_VEL
LIN {X 0,Y 531.045,Z 710.409,A -85,B 0,C 180,E1 -4279.249,E2 -4279.249} C_VEL
LIN {X 0,Y 532.117,Z 714.657,A -85,B 0,C 180,E1 -4279.47,E2 -4279.47} C_VEL
LIN {X 0,Y 531.95,Z 725.308,A -85,B 0,C 180,E1 -4280.022,E2 -4280.022} C_VEL
LIN {X 0,Y 531.709,Z 734.62,A -85,B 0,C 180,E1 -4280.62,E2 -4280.62} C_VEL
LIN {X 0,Y 531.484,Z 744.039,A -85,B 0,C 180,E1 -4281.361,E2 -4281.361} C_VEL
LIN {X 0,Y 531.321,Z 752.465,A -85,B 0,C 180,E1 -4282.162,E2 -4282.162} C_VEL
LIN {X 0,Y 531.133,Z 759.706,A -85,B 0,C 180,E1 -4282.982,E2 -4282.982} C_VEL
LIN {X 0,Y 530.917,Z 766.208,A -85,B 0,C 180,E1 -4283.852,E2 -4283.852} C_VEL
LIN {X 0,Y 530.829,Z 772.239,A -85,B 0,C 180,E1 -4284.818,E2 -4284.818} C_VEL
LIN {X 0,Y 530.703,Z 777.089,A -85,B 0,C 180,E1 -4285.749,E2 -4285.749} C_VEL
LIN {X 0,Y 530.582,Z 781.664,A -85,B 0,C 180,E1 -4286.828,E2 -4286.828} C_VEL
LIN {X 0,Y 530.529,Z 785.521,A -85,B 0,C 180,E1 -4288.002,E2 -4288.002} C_VEL
LIN {X 0,Y 530.5,Z 787.765,A -85,B 0,C 180,E1 -4288.891,E2 -4288.891} C_VEL
LIN {X 0,Y 530.486,Z 789.44,A -85,B 0,C 180,E1 -4289.772,E2 -4289.772} C_VEL
LIN {X 0,Y 530.458,Z 790.8,A -85,B 0,C 180,E1 -4290.978,E2 -4290.978} C_VEL
LIN {X 0,Y 530.435,Z 791.035,A -85,B 0,C 180,E1 -4292.588,E2 -4292.588} C_VEL
LIN {X 0,Y 530.46,Z 790.745,A -85,B 0,C 180,E1 -4293.226,E2 -4293.226} C_VEL
LIN {X 0,Y 530.462,Z 789.54,A -85,B 0,C 180,E1 -4294.28,E2 -4294.28} C_VEL
LIN {X 0,Y 530.558,Z 786.541,A -85,B 0,C 180,E1 -4295.755,E2 -4295.755} C_VEL
LIN {X 0,Y 530.6,Z 782.755,A -85,B 0,C 180,E1 -4296.999,E2 -4296.999} C_VEL
LIN {X 0,Y 530.683,Z 778.918,A -85,B 0,C 180,E1 -4297.978,E2 -4297.978} C_VEL
LIN {X 0,Y 530.805,Z 773.659,A -85,B 0,C 180,E1 -4299.054,E2 -4299.054} C_VEL
LIN {X 0,Y 530.97,Z 767.128,A -85,B 0,C 180,E1 -4300.135,E2 -4300.135} C_VEL
LIN {X 0,Y 531.141,Z 760.175,A -85,B 0,C 180,E1 -4301.084,E2 -4301.084} C_VEL
LIN {X 0,Y 531.361,Z 752.07,A -85,B 0,C 180,E1 -4302.001,E2 -4302.001} C_VEL
LIN {X 0,Y 531.552,Z 743.661,A -85,B 0,C 180,E1 -4302.792,E2 -4302.792} C_VEL
LIN {X 0,Y 531.799,Z 733.315,A -85,B 0,C 180,E1 -4303.591,E2 -4303.591} C_VEL
LIN {X 0,Y 532.019,Z 722.341,A -85,B 0,C 180,E1 -4304.265,E2 -4304.265} C_VEL
LIN {X 0,Y 531.954,Z 714.012,A -85,B 0,C 180,E1 -4304.678,E2 -4304.678} C_VEL
LIN {X 0,Y 531.031,Z 710.337,A -85,B 0,C 180,E1 -4304.879,E2 -4304.879} C_VEL
LIN {X 0,Y 531.054,Z 710.333,A -85,B 0,C 180,E1 -4308.329,E2 -4308.329} C_VEL
LIN {X 0,Y 531.055,Z 710.339,A -85,B 0,C 180,E1 -4311.629,E2 -4311.629} C_VEL
LIN {X 0,Y 531.111,Z 710.322,A -85,B 0,C 180,E1 -4314.685,E2 -4314.685} C_VEL
LIN {X 0,Y 531.142,Z 710.328,A -85,B 0,C 180,E1 -4317.725,E2 -4317.725} C_VEL
LIN {X 0,Y 531.154,Z 710.317,A -85,B 0,C 180,E1 -4320.758,E2 -4320.758} C_VEL
LIN {X 0,Y 531.105,Z 710.322,A -85,B 0,C 180,E1 -4323.034,E2 -4323.034} C_VEL
LIN {X 0,Y 531.086,Z 710.332,A -85,B 0,C 180,E1 -4326.077,E2 -4326.077} C_VEL
LIN {X 0,Y 531.02,Z 710.332,A -85,B 0,C 180,E1 -4329.138,E2 -4329.138} C_VEL
LIN {X 0,Y 531.044,Z 710.337,A -85,B 0,C 180,E1 -4332.225,E2 -4332.225} C_VEL
LIN {X 0,Y 531,Z 710.334,A -85,B 0,C 180,E1 -4335.35,E2 -4335.35} C_VEL
LIN {X 0,Y 530.99,Z 710.342,A -85,B 0,C 180,E1 -4338.521,E2 -4338.521} C_VEL
LIN {X 0,Y 531.003,Z 710.335,A -85,B 0,C 180,E1 -4340.938,E2 -4340.938} C_VEL
LIN {X 0,Y 530.969,Z 710.347,A -85,B 0,C 180,E1 -4344.225,E2 -4344.225} C_VEL
LIN {X 0,Y 531.005,Z 710.339,A -85,B 0,C 180,E1 -4346.744,E2 -4346.744} C_VEL
LIN {X 0,Y 530.986,Z 710.338,A -85,B 0,C 180,E1 -4349.322,E2 -4349.322} C_VEL
LIN {X 0,Y 530.974,Z 710.344,A -85,B 0,C 180,E1 -4352.101,E2 -4352.101} C_VEL
LIN {X 0,Y 530.976,Z 710.344,A -85,B 0,C 180,E1 -4354.851,E2 -4354.851} C_VEL
LIN {X 0,Y 530.969,Z 710.342,A -85,B 0,C 180,E1 -4357.507,E2 -4357.507} C_VEL
LIN {X 0,Y 530.987,Z 710.347,A -85,B 0,C 180,E1 -4360.433,E2 -4360.433} C_VEL
LIN {X 0,Y 530.968,Z 710.342,A -85,B 0,C 180,E1 -4363.494,E2 -4363.494} C_VEL
LIN {X 0,Y 530.964,Z 710.349,A -85,B 0,C 180,E1 -4366.505,E2 -4366.505} C_VEL
LIN {X 0,Y 530.992,Z 710.347,A -85,B 0,C 180,E1 -4368.976,E2 -4368.976} C_VEL
LIN {X 0,Y 530.995,Z 710.498,A -85,B 0,C 180,E1 -4371.955,E2 -4371.955} C_VEL
LIN {X 0,Y 532.368,Z 717.495,A -85,B 0,C 180,E1 -4373.638,E2 -4373.638} C_VEL
LIN {X 0,Y 532.577,Z 721.372,A -85,B 0,C 180,E1 -4374.505,E2 -4374.505} C_VEL
LIN {X 0,Y 532.401,Z 735.346,A -85,B 0,C 180,E1 -4377.489,E2 -4377.489} C_VEL
LIN {X 0,Y 532.249,Z 748.094,A -85,B 0,C 180,E1 -4380.093,E2 -4380.093} C_VEL
LIN {X 0,Y 532.104,Z 764.351,A -85,B 0,C 180,E1 -4383.316,E2 -4383.316} C_VEL
LIN {X 0,Y 531.925,Z 778.354,A -85,B 0,C 180,E1 -4386.028,E2 -4386.028} C_VEL
LIN {X 0,Y 531.776,Z 788.485,A -85,B 0,C 180,E1 -4387.981,E2 -4387.981} C_VEL
LIN {X 0,Y 531.456,Z 801.665,A -85,B 0,C 180,E1 -4390.695,E2 -4390.695} C_VEL
LIN {X 0,Y 531.2,Z 815.36,A -85,B 0,C 180,E1 -4393.474,E2 -4393.474} C_VEL
LIN {X 0,Y 530.931,Z 830.156,A -85,B 0,C 180,E1 -4396.435,E2 -4396.435} C_VEL
LIN {X 0,Y 532.382,Z 840.501,A -85,B 0,C 180,E1 -4396.667,E2 -4396.667} C_VEL
LIN {X 0,Y 532.174,Z 852.87,A -85,B 0,C 180,E1 -4397.026,E2 -4397.026} C_VEL
LIN {X 0,Y 531.975,Z 864.502,A -85,B 0,C 180,E1 -4397.506,E2 -4397.506} C_VEL
LIN {X 0,Y 531.77,Z 876.095,A -85,B 0,C 180,E1 -4398.137,E2 -4398.137} C_VEL
LIN {X 0,Y 531.528,Z 886.483,A -85,B 0,C 180,E1 -4398.85,E2 -4398.85} C_VEL
LIN {X 0,Y 531.224,Z 896.645,A -85,B 0,C 180,E1 -4399.711,E2 -4399.711} C_VEL
LIN {X 0,Y 531.012,Z 905.785,A -85,B 0,C 180,E1 -4400.669,E2 -4400.669} C_VEL
LIN {X 0,Y 530.813,Z 914.688,A -85,B 0,C 180,E1 -4401.817,E2 -4401.817} C_VEL
LIN {X 0,Y 530.664,Z 921.848,A -85,B 0,C 180,E1 -4402.963,E2 -4402.963} C_VEL
LIN {X 0,Y 530.611,Z 928.365,A -85,B 0,C 180,E1 -4404.299,E2 -4404.299} C_VEL
LIN {X 0,Y 530.457,Z 932.677,A -85,B 0,C 180,E1 -4405.44,E2 -4405.44} C_VEL
LIN {X 0,Y 530.516,Z 934.958,A -85,B 0,C 180,E1 -4406.202,E2 -4406.202} C_VEL
LIN {X 0,Y 530.457,Z 936.807,A -85,B 0,C 180,E1 -4406.962,E2 -4406.962} C_VEL
LIN {X 0,Y 530.41,Z 938.196,A -85,B 0,C 180,E1 -4407.722,E2 -4407.722} C_VEL
LIN {X 0,Y 530.344,Z 939.786,A -85,B 0,C 180,E1 -4409.241,E2 -4409.241} C_VEL
LIN {X 0,Y 530.342,Z 940,A -85,B 0,C 180,E1 -4410,E2 -4410} C_VEL
LIN {X 0,Y 530.361,Z 939.185,A -85,B 0,C 180,E1 -4411.519,E2 -4411.519} C_VEL
LIN {X 0,Y 530.41,Z 938.198,A -85,B 0,C 180,E1 -4412.278,E2 -4412.278} C_VEL
LIN {X 0,Y 530.457,Z 936.81,A -85,B 0,C 180,E1 -4413.038,E2 -4413.038} C_VEL
LIN {X 0,Y 530.522,Z 933.896,A -85,B 0,C 180,E1 -4414.178,E2 -4414.178} C_VEL
LIN {X 0,Y 530.524,Z 929.949,A -85,B 0,C 180,E1 -4415.321,E2 -4415.321} C_VEL
LIN {X 0,Y 530.599,Z 924.263,A -85,B 0,C 180,E1 -4416.582,E2 -4416.582} C_VEL
LIN {X 0,Y 530.758,Z 917.237,A -85,B 0,C 180,E1 -4417.8,E2 -4417.8} C_VEL
LIN {X 0,Y 530.931,Z 908.992,A -85,B 0,C 180,E1 -4418.948,E2 -4418.948} C_VEL
LIN {X 0,Y 531.112,Z 900.539,A -85,B 0,C 180,E1 -4419.905,E2 -4419.905} C_VEL
LIN {X 0,Y 531.421,Z 890.095,A -85,B 0,C 180,E1 -4420.863,E2 -4420.863} C_VEL
LIN {X 0,Y 531.646,Z 879.3,A -85,B 0,C 180,E1 -4421.661,E2 -4421.661} C_VEL
LIN {X 0,Y 531.871,Z 868.407,A -85,B 0,C 180,E1 -4422.302,E2 -4422.302} C_VEL
LIN {X 0,Y 532.112,Z 856.764,A -85,B 0,C 180,E1 -4422.83,E2 -4422.83} C_VEL
LIN {X 0,Y 532.33,Z 843.346,A -85,B 0,C 180,E1 -4423.261,E2 -4423.261} C_VEL
LIN {X 0,Y 532.13,Z 837.787,A -85,B 0,C 180,E1 -4423.397,E2 -4423.397} C_VEL
LIN {X 0,Y 530.943,Z 830.034,A -85,B 0,C 180,E1 -4423.589,E2 -4423.589} C_VEL
LIN {X 0,Y 531.2,Z 815.361,A -85,B 0,C 180,E1 -4426.526,E2 -4426.526} C_VEL
LIN {X 0,Y 531.456,Z 801.666,A -85,B 0,C 180,E1 -4429.305,E2 -4429.305} C_VEL
LIN {X 0,Y 531.775,Z 788.486,A -85,B 0,C 180,E1 -4432.019,E2 -4432.019} C_VEL
LIN {X 0,Y 532.045,Z 773.319,A -85,B 0,C 180,E1 -4435.005,E2 -4435.005} C_VEL
LIN {X 0,Y 532.251,Z 759.697,A -85,B 0,C 180,E1 -4437.787,E2 -4437.787} C_VEL
LIN {X 0,Y 532.527,Z 746.527,A -85,B 0,C 180,E1 -4440.518,E2 -4440.518} C_VEL
LIN {X 0,Y 532.839,Z 731.994,A -85,B 0,C 180,E1 -4443.64,E2 -4443.64} C_VEL
LIN {X 0,Y 532.989,Z 720.764,A -85,B 0,C 180,E1 -4446.162,E2 -4446.162} C_VEL
LIN {X 0,Y 531.411,Z 712.493,A -85,B 0,C 180,E1 -4448.197,E2 -4448.197} C_VEL
LIN {X 0,Y 530.975,Z 710.347,A -85,B 0,C 180,E1 -4448.749,E2 -4448.749} C_VEL
LIN {X 0,Y 531.003,Z 710.345,A -85,B 0,C 180,E1 -4451.435,E2 -4451.435} C_VEL
LIN {X 0,Y 530.99,Z 710.339,A -85,B 0,C 180,E1 -4454.547,E2 -4454.547} C_VEL
LIN {X 0,Y 530.986,Z 710.342,A -85,B 0,C 180,E1 -4457.834,E2 -4457.834} C_VEL
LIN {X 0,Y 530.993,Z 710.337,A -85,B 0,C 180,E1 -4460.557,E2 -4460.557} C_VEL
LIN {X 0,Y 530.958,Z 710.35,A -85,B 0,C 180,E1 -4463.442,E2 -4463.442} C_VEL
LIN {X 0,Y 531.002,Z 710.336,A -85,B 0,C 180,E1 -4466.494,E2 -4466.494} C_VEL
LIN {X 0,Y 530.977,Z 710.345,A -85,B 0,C 180,E1 -4469.355,E2 -4469.355} C_VEL
LIN {X 0,Y 531.015,Z 710.334,A -85,B 0,C 180,E1 -4472.468,E2 -4472.468} C_VEL
LIN {X 0,Y 530.997,Z 710.337,A -85,B 0,C 180,E1 -4474.942,E2 -4474.942} C_VEL
LIN {X 0,Y 530.974,Z 710.342,A -85,B 0,C 180,E1 -4478.247,E2 -4478.247} C_VEL
LIN {X 0,Y 530.995,Z 710.337,A -85,B 0,C 180,E1 -4480.677,E2 -4480.677} C_VEL
LIN {X 0,Y 530.978,Z 710.34,A -85,B 0,C 180,E1 -4483.071,E2 -4483.071} C_VEL
LIN {X 0,Y 531.022,Z 710.337,A -85,B 0,C 180,E1 -4485.436,E2 -4485.436} C_VEL
LIN {X 0,Y 531.04,Z 710.333,A -85,B 0,C 180,E1 -4488.55,E2 -4488.55} C_VEL
LIN {X 0,Y 531.055,Z 710.334,A -85,B 0,C 180,E1 -4491.629,E2 -4491.629} C_VEL
LIN {X 0,Y 531.12,Z 710.323,A -85,B 0,C 180,E1 -4494.685,E2 -4494.685} C_VEL
LIN {X 0,Y 531.142,Z 710.323,A -85,B 0,C 180,E1 -4497.725,E2 -4497.725} C_VEL
LIN {X 0,Y 531.149,Z 710.32,A -85,B 0,C 180,E1 -4500.758,E2 -4500.758} C_VEL
LIN {X 0,Y 531.099,Z 710.325,A -85,B 0,C 180,E1 -4503.034,E2 -4503.034} C_VEL
LIN {X 0,Y 531.067,Z 710.335,A -85,B 0,C 180,E1 -4506.077,E2 -4506.077} C_VEL
LIN {X 0,Y 531.019,Z 710.335,A -85,B 0,C 180,E1 -4509.138,E2 -4509.138} C_VEL
LIN {X 0,Y 531.052,Z 710.332,A -85,B 0,C 180,E1 -4511.671,E2 -4511.671} C_VEL
LIN {X 0,Y 531.026,Z 710.336,A -85,B 0,C 180,E1 -4514.952,E2 -4514.952} C_VEL
LIN {X 0,Y 530.983,Z 710.34,A -85,B 0,C 180,E1 -4517.724,E2 -4517.724} C_VEL
LIN {X 0,Y 531.028,Z 710.338,A -85,B 0,C 180,E1 -4520.127,E2 -4520.127} C_VEL
LIN {X 0,Y 530.946,Z 710.351,A -85,B 0,C 180,E1 -4522.574,E2 -4522.574} C_VEL
LIN {X 0,Y 530.949,Z 710.346,A -85,B 0,C 180,E1 -4525.061,E2 -4525.061} C_VEL
LIN {X 0,Y 530.964,Z 710.341,A -85,B 0,C 180,E1 -4527.599,E2 -4527.599} C_VEL
LIN {X 0,Y 530.954,Z 710.346,A -85,B 0,C 180,E1 -4530.198,E2 -4530.198} C_VEL
LIN {X 0,Y 530.969,Z 710.348,A -85,B 0,C 180,E1 -4532.867,E2 -4532.867} C_VEL
LIN {X 0,Y 530.949,Z 710.344,A -85,B 0,C 180,E1 -4535.621,E2 -4535.621} C_VEL
LIN {X 0,Y 530.959,Z 710.349,A -85,B 0,C 180,E1 -4538.652,E2 -4538.652} C_VEL
LIN {X 0,Y 530.954,Z 710.344,A -85,B 0,C 180,E1 -4541.44,E2 -4541.44} C_VEL
LIN {X 0,Y 530.927,Z 710.347,A -85,B 0,C 180,E1 -4543.543,E2 -4543.543} C_VEL
LIN {X 0,Y 530.263,Z 710.43,A -85,B 0,C 180,E1 -4544.177,E2 -4544.177} C_VEL
LIN {X 0,Y 527.424,Z 710.789,A -85,B 0,C 180,E1 -4545.206,E2 -4545.206} C_VEL
LIN {X 0,Y 525.016,Z 711.093,A -85,B 0,C 180,E1 -4546.035,E2 -4546.035} C_VEL
LIN {X 0,Y 523.97,Z 711.221,A -85,B 0,C 180,E1 -4546.674,E2 -4546.674} C_VEL
LIN {X 0,Y 523.879,Z 711.23,A -85,B 0,C 180,E1 -4546.891,E2 -4546.891} C_VEL
LIN {X 0,Y 523.915,Z 711.22,A -85,B 0,C 180,E1 -4549.917,E2 -4549.917} C_VEL
LIN {X 0,Y 523.876,Z 711.232,A -85,B 0,C 180,E1 -4552.865,E2 -4552.865} C_VEL
LIN {X 0,Y 523.906,Z 711.222,A -85,B 0,C 180,E1 -4555.708,E2 -4555.708} C_VEL
LIN {X 0,Y 523.907,Z 711.222,A -85,B 0,C 180,E1 -4558.455,E2 -4558.455} C_VEL
LIN {X 0,Y 523.9,Z 711.228,A -85,B 0,C 180,E1 -4561.123,E2 -4561.123} C_VEL
LIN {X 0,Y 523.879,Z 711.225,A -85,B 0,C 180,E1 -4564.005,E2 -4564.005} C_VEL
LIN {X 0,Y 523.909,Z 711.22,A -85,B 0,C 180,E1 -4566.269,E2 -4566.269} C_VEL
LIN {X 0,Y 523.946,Z 711.218,A -85,B 0,C 180,E1 -4568.767,E2 -4568.767} C_VEL
LIN {X 0,Y 523.936,Z 711.225,A -85,B 0,C 180,E1 -4571.22,E2 -4571.22} C_VEL
LIN {X 0,Y 523.893,Z 711.228,A -85,B 0,C 180,E1 -4573.637,E2 -4573.637} C_VEL
LIN {X 0,Y 523.918,Z 711.221,A -85,B 0,C 180,E1 -4576.027,E2 -4576.027} C_VEL
LIN {X 0,Y 523.965,Z 711.213,A -85,B 0,C 180,E1 -4578.393,E2 -4578.393} C_VEL
LIN {X 0,Y 523.947,Z 711.223,A -85,B 0,C 180,E1 -4581.515,E2 -4581.515} C_VEL
LIN {X 0,Y 524.032,Z 711.205,A -85,B 0,C 180,E1 -4584.613,E2 -4584.613} C_VEL
LIN {X 0,Y 524.106,Z 711.202,A -85,B 0,C 180,E1 -4587.695,E2 -4587.695} C_VEL
LIN {X 0,Y 524.1,Z 711.201,A -85,B 0,C 180,E1 -4590,E2 -4590} C_VEL
LIN {X 0,Y 524.107,Z 711.197,A -85,B 0,C 180,E1 -4592.306,E2 -4592.306} C_VEL
LIN {X 0,Y 524.012,Z 711.211,A -85,B 0,C 180,E1 -4596.16,E2 -4596.16} C_VEL
LIN {X 0,Y 523.984,Z 711.212,A -85,B 0,C 180,E1 -4599.262,E2 -4599.262} C_VEL
LIN {X 0,Y 524.003,Z 711.215,A -85,B 0,C 180,E1 -4601.737,E2 -4601.737} C_VEL
LIN {X 0,Y 523.998,Z 711.209,A -85,B 0,C 180,E1 -4605.052,E2 -4605.052} C_VEL
LIN {X 0,Y 523.949,Z 711.223,A -85,B 0,C 180,E1 -4607.97,E2 -4607.97} C_VEL
LIN {X 0,Y 523.976,Z 711.216,A -85,B 0,C 180,E1 -4610.41,E2 -4610.41} C_VEL
LIN {X 0,Y 523.914,Z 711.219,A -85,B 0,C 180,E1 -4612.894,E2 -4612.894} C_VEL
LIN {X 0,Y 523.908,Z 711.221,A -85,B 0,C 180,E1 -4615.421,E2 -4615.421} C_VEL
LIN {X 0,Y 523.919,Z 711.225,A -85,B 0,C 180,E1 -4618.002,E2 -4618.002} C_VEL
LIN {X 0,Y 523.944,Z 711.217,A -85,B 0,C 180,E1 -4620.854,E2 -4620.854} C_VEL
LIN {X 0,Y 523.934,Z 711.218,A -85,B 0,C 180,E1 -4623.73,E2 -4623.73} C_VEL
LIN {X 0,Y 523.908,Z 711.227,A -85,B 0,C 180,E1 -4626.401,E2 -4626.401} C_VEL
LIN {X 0,Y 523.924,Z 711.218,A -85,B 0,C 180,E1 -4629.085,E2 -4629.085} C_VEL
LIN {X 0,Y 523.955,Z 711.218,A -85,B 0,C 180,E1 -4632.119,E2 -4632.119} C_VEL
LIN {X 0,Y 523.946,Z 711.216,A -85,B 0,C 180,E1 -4635.31,E2 -4635.31} C_VEL
LIN {X 0,Y 523.967,Z 711.221,A -85,B 0,C 180,E1 -4638.689,E2 -4638.689} C_VEL
LIN {X 0,Y 523.973,Z 711.217,A -85,B 0,C 180,E1 -4639.072,E2 -4639.072} C_VEL
LIN {X 0,Y 525.268,Z 716.205,A -85,B 0,C 180,E1 -4639.338,E2 -4639.338} C_VEL
LIN {X 0,Y 525.061,Z 727.025,A -85,B 0,C 180,E1 -4639.914,E2 -4639.914} C_VEL
LIN {X 0,Y 524.78,Z 737.567,A -85,B 0,C 180,E1 -4640.62,E2 -4640.62} C_VEL
LIN {X 0,Y 524.553,Z 747.685,A -85,B 0,C 180,E1 -4641.463,E2 -4641.463} C_VEL
LIN {X 0,Y 524.283,Z 757.463,A -85,B 0,C 180,E1 -4642.472,E2 -4642.472} C_VEL
LIN {X 0,Y 524.012,Z 766.086,A -85,B 0,C 180,E1 -4643.583,E2 -4643.583} C_VEL
LIN {X 0,Y 523.888,Z 772.162,A -85,B 0,C 180,E1 -4644.535,E2 -4644.535} C_VEL
LIN {X 0,Y 523.71,Z 778.201,A -85,B 0,C 180,E1 -4645.693,E2 -4645.693} C_VEL
LIN {X 0,Y 523.614,Z 782.123,A -85,B 0,C 180,E1 -4646.612,E2 -4646.612} C_VEL
LIN {X 0,Y 523.543,Z 785.978,A -85,B 0,C 180,E1 -4647.748,E2 -4647.748} C_VEL
LIN {X 0,Y 523.557,Z 787.851,A -85,B 0,C 180,E1 -4648.431,E2 -4648.431} C_VEL
LIN {X 0,Y 523.472,Z 789.708,A -85,B 0,C 180,E1 -4649.324,E2 -4649.324} C_VEL
LIN {X 0,Y 523.431,Z 791.689,A -85,B 0,C 180,E1 -4650.78,E2 -4650.78} C_VEL
LIN {X 0,Y 523.419,Z 792.166,A -85,B 0,C 180,E1 -4652.399,E2 -4652.399} C_VEL
LIN {X 0,Y 523.449,Z 790.857,A -85,B 0,C 180,E1 -4654.102,E2 -4654.102} C_VEL
LIN {X 0,Y 523.524,Z 788.557,A -85,B 0,C 180,E1 -4655.408,E2 -4655.408} C_VEL
LIN {X 0,Y 523.611,Z 785.162,A -85,B 0,C 180,E1 -4656.674,E2 -4656.674} C_VEL
LIN {X 0,Y 523.72,Z 780.556,A -85,B 0,C 180,E1 -4657.93,E2 -4657.93} C_VEL
LIN {X 0,Y 523.85,Z 774.577,A -85,B 0,C 180,E1 -4659.174,E2 -4659.174} C_VEL
LIN {X 0,Y 524.025,Z 768.871,A -85,B 0,C 180,E1 -4660.141,E2 -4660.141} C_VEL
LIN {X 0,Y 524.243,Z 761.013,A -85,B 0,C 180,E1 -4661.231,E2 -4661.231} C_VEL
LIN {X 0,Y 524.474,Z 752.458,A -85,B 0,C 180,E1 -4662.204,E2 -4662.204} C_VEL
LIN {X 0,Y 524.766,Z 742.018,A -85,B 0,C 180,E1 -4663.165,E2 -4663.165} C_VEL
LIN {X 0,Y 524.959,Z 730.991,A -85,B 0,C 180,E1 -4663.971,E2 -4663.971} C_VEL
LIN {X 0,Y 525.237,Z 719.229,A -85,B 0,C 180,E1 -4664.638,E2 -4664.638} C_VEL
LIN {X 0,Y 525.207,Z 715.966,A -85,B 0,C 180,E1 -4664.797,E2 -4664.797} C_VEL
LIN {X 0,Y 523.997,Z 711.216,A -85,B 0,C 180,E1 -4665.062,E2 -4665.062} C_VEL
LIN {X 0,Y 524.018,Z 711.21,A -85,B 0,C 180,E1 -4668.394,E2 -4668.394} C_VEL
LIN {X 0,Y 524.003,Z 711.216,A -85,B 0,C 180,E1 -4671.516,E2 -4671.516} C_VEL
LIN {X 0,Y 524.071,Z 711.199,A -85,B 0,C 180,E1 -4674.613,E2 -4674.613} C_VEL
LIN {X 0,Y 524.114,Z 711.203,A -85,B 0,C 180,E1 -4677.694,E2 -4677.694} C_VEL
LIN {X 0,Y 524.125,Z 711.193,A -85,B 0,C 180,E1 -4680.768,E2 -4680.768} C_VEL
LIN {X 0,Y 524.046,Z 711.201,A -85,B 0,C 180,E1 -4683.075,E2 -4683.075} C_VEL
LIN {X 0,Y 524.048,Z 711.208,A -85,B 0,C 180,E1 -4686.159,E2 -4686.159} C_VEL
LIN {X 0,Y 523.99,Z 711.208,A -85,B 0,C 180,E1 -4689.262,E2 -4689.262} C_VEL
LIN {X 0,Y 524.008,Z 711.212,A -85,B 0,C 180,E1 -4691.739,E2 -4691.739} C_VEL
LIN {X 0,Y 523.998,Z 711.206,A -85,B 0,C 180,E1 -4695.052,E2 -4695.052} C_VEL
LIN {X 0,Y 523.952,Z 711.221,A -85,B 0,C 180,E1 -4697.969,E2 -4697.969} C_VEL
LIN {X 0,Y 523.976,Z 711.216,A -85,B 0,C 180,E1 -4700.41,E2 -4700.41} C_VEL
LIN {X 0,Y 523.914,Z 711.22,A -85,B 0,C 180,E1 -4702.893,E2 -4702.893} C_VEL
LIN {X 0,Y 523.988,Z 711.215,A -85,B 0,C 180,E1 -4706.02,E2 -4706.02} C_VEL
LIN {X 0,Y 523.943,Z 711.218,A -85,B 0,C 180,E1 -4708.875,E2 -4708.875} C_VEL
LIN {X 0,Y 523.927,Z 711.217,A -85,B 0,C 180,E1 -4711.544,E2 -4711.544} C_VEL
LIN {X 0,Y 523.938,Z 711.223,A -85,B 0,C 180,E1 -4714.29,E2 -4714.29} C_VEL
LIN {X 0,Y 523.911,Z 711.223,A -85,B 0,C 180,E1 -4717.132,E2 -4717.132} C_VEL
LIN {X 0,Y 523.941,Z 711.222,A -85,B 0,C 180,E1 -4720.13,E2 -4720.13} C_VEL
LIN {X 0,Y 523.939,Z 711.224,A -85,B 0,C 180,E1 -4722.459,E2 -4722.459} C_VEL
LIN {X 0,Y 523.959,Z 711.216,A -85,B 0,C 180,E1 -4725.309,E2 -4725.309} C_VEL
LIN {X 0,Y 523.965,Z 711.222,A -85,B 0,C 180,E1 -4728.689,E2 -4728.689} C_VEL
LIN {X 0,Y 523.97,Z 711.35,A -85,B 0,C 180,E1 -4731.719,E2 -4731.719} C_VEL
LIN {X 0,Y 525.645,Z 720.573,A -85,B 0,C 180,E1 -4733.964,E2 -4733.964} C_VEL
LIN {X 0,Y 525.48,Z 733.227,A -85,B 0,C 180,E1 -4736.746,E2 -4736.746} C_VEL
LIN {X 0,Y 525.258,Z 747.141,A -85,B 0,C 180,E1 -4739.662,E2 -4739.662} C_VEL
LIN {X 0,Y 525.052,Z 762.252,A -85,B 0,C 180,E1 -4742.713,E2 -4742.713} C_VEL
LIN {X 0,Y 524.896,Z 776.62,A -85,B 0,C 180,E1 -4745.571,E2 -4745.571} C_VEL
LIN {X 0,Y 524.674,Z 791.327,A -85,B 0,C 180,E1 -4748.385,E2 -4748.385} C_VEL
LIN {X 0,Y 524.486,Z 801.665,A -85,B 0,C 180,E1 -4750.428,E2 -4750.428} C_VEL
LIN {X 0,Y 524.181,Z 815.36,A -85,B 0,C 180,E1 -4753.246,E2 -4753.246} C_VEL
LIN {X 0,Y 523.898,Z 830.156,A -85,B 0,C 180,E1 -4756.249,E2 -4756.249} C_VEL
LIN {X 0,Y 525.459,Z 841.514,A -85,B 0,C 180,E1 -4756.513,E2 -4756.513} C_VEL
LIN {X 0,Y 525.256,Z 854.17,A -85,B 0,C 180,E1 -4756.901,E2 -4756.901} C_VEL
LIN {X 0,Y 524.986,Z 866.488,A -85,B 0,C 180,E1 -4757.435,E2 -4757.435} C_VEL
LIN {X 0,Y 524.766,Z 878.28,A -85,B 0,C 180,E1 -4758.114,E2 -4758.114} C_VEL
LIN {X 0,Y 524.493,Z 888.919,A -85,B 0,C 180,E1 -4758.894,E2 -4758.894} C_VEL
LIN {X 0,Y 524.167,Z 898.597,A -85,B 0,C 180,E1 -4759.767,E2 -4759.767} C_VEL
LIN {X 0,Y 523.929,Z 907.412,A -85,B 0,C 180,E1 -4760.737,E2 -4760.737} C_VEL
LIN {X 0,Y 523.724,Z 916.002,A -85,B 0,C 180,E1 -4761.9,E2 -4761.9} C_VEL
LIN {X 0,Y 523.575,Z 922.868,A -85,B 0,C 180,E1 -4763.061,E2 -4763.061} C_VEL
LIN {X 0,Y 523.544,Z 928.365,A -85,B 0,C 180,E1 -4764.222,E2 -4764.222} C_VEL
LIN {X 0,Y 523.361,Z 932.677,A -85,B 0,C 180,E1 -4765.378,E2 -4765.378} C_VEL
LIN {X 0,Y 523.443,Z 934.958,A -85,B 0,C 180,E1 -4766.151,E2 -4766.151} C_VEL
LIN {X 0,Y 523.368,Z 936.807,A -85,B 0,C 180,E1 -4766.921,E2 -4766.921} C_VEL
LIN {X 0,Y 523.334,Z 938.195,A -85,B 0,C 180,E1 -4767.691,E2 -4767.691} C_VEL
LIN {X 0,Y 523.25,Z 939.786,A -85,B 0,C 180,E1 -4769.23,E2 -4769.23} C_VEL
LIN {X 0,Y 523.246,Z 940,A -85,B 0,C 180,E1 -4770,E2 -4770} C_VEL
LIN {X 0,Y 523.274,Z 939.185,A -85,B 0,C 180,E1 -4771.539,E2 -4771.539} C_VEL
LIN {X 0,Y 523.334,Z 938.197,A -85,B 0,C 180,E1 -4772.309,E2 -4772.309} C_VEL
LIN {X 0,Y 523.368,Z 936.81,A -85,B 0,C 180,E1 -4773.079,E2 -4773.079} C_VEL
LIN {X 0,Y 523.441,Z 933.896,A -85,B 0,C 180,E1 -4774.235,E2 -4774.235} C_VEL
LIN {X 0,Y 523.464,Z 929.949,A -85,B 0,C 180,E1 -4775.393,E2 -4775.393} C_VEL
LIN {X 0,Y 523.523,Z 924.727,A -85,B 0,C 180,E1 -4776.581,E2 -4776.581} C_VEL
LIN {X 0,Y 523.665,Z 918.467,A -85,B 0,C 180,E1 -4777.713,E2 -4777.713} C_VEL
LIN {X 0,Y 523.857,Z 910.478,A -85,B 0,C 180,E1 -4778.875,E2 -4778.875} C_VEL
LIN {X 0,Y 524.084,Z 902.334,A -85,B 0,C 180,E1 -4779.845,E2 -4779.845} C_VEL
LIN {X 0,Y 524.355,Z 892.399,A -85,B 0,C 180,E1 -4780.815,E2 -4780.815} C_VEL
LIN {X 0,Y 524.684,Z 881.132,A -85,B 0,C 180,E1 -4781.692,E2 -4781.692} C_VEL
LIN {X 0,Y 524.9,Z 870.173,A -85,B 0,C 180,E1 -4782.37,E2 -4782.37} C_VEL
LIN {X 0,Y 525.177,Z 857.975,A -85,B 0,C 180,E1 -4782.953,E2 -4782.953} C_VEL
LIN {X 0,Y 525.42,Z 845.174,A -85,B 0,C 180,E1 -4783.39,E2 -4783.39} C_VEL
LIN {X 0,Y 525.255,Z 838.667,A -85,B 0,C 180,E1 -4783.557,E2 -4783.557} C_VEL
LIN {X 0,Y 523.894,Z 830.034,A -85,B 0,C 180,E1 -4783.775,E2 -4783.775} C_VEL
LIN {X 0,Y 524.18,Z 815.361,A -85,B 0,C 180,E1 -4786.754,E2 -4786.754} C_VEL
LIN {X 0,Y 524.485,Z 801.666,A -85,B 0,C 180,E1 -4789.572,E2 -4789.572} C_VEL
LIN {X 0,Y 524.72,Z 789.34,A -85,B 0,C 180,E1 -4792.026,E2 -4792.026} C_VEL
LIN {X 0,Y 525.014,Z 774.738,A -85,B 0,C 180,E1 -4794.94,E2 -4794.94} C_VEL
LIN {X 0,Y 525.277,Z 760.012,A -85,B 0,C 180,E1 -4797.987,E2 -4797.987} C_VEL
LIN {X 0,Y 525.627,Z 745.055,A -85,B 0,C 180,E1 -4801.16,E2 -4801.16} C_VEL
LIN {X 0,Y 525.935,Z 731.87,A -85,B 0,C 180,E1 -4804.055,E2 -4804.055} C_VEL
LIN {X 0,Y 526.079,Z 721.92,A -85,B 0,C 180,E1 -4806.336,E2 -4806.336} C_VEL
LIN {X 0,Y 523.937,Z 711.225,A -85,B 0,C 180,E1 -4809.027,E2 -4809.027} C_VEL
LIN {X 0,Y 523.96,Z 711.216,A -85,B 0,C 180,E1 -4812.118,E2 -4812.118} C_VEL
LIN {X 0,Y 523.959,Z 711.221,A -85,B 0,C 180,E1 -4815.309,E2 -4815.309} C_VEL
LIN {X 0,Y 523.962,Z 711.215,A -85,B 0,C 180,E1 -4818.689,E2 -4818.689} C_VEL
LIN {X 0,Y 523.919,Z 711.221,A -85,B 0,C 180,E1 -4821.898,E2 -4821.898} C_VEL
LIN {X 0,Y 523.928,Z 711.219,A -85,B 0,C 180,E1 -4824.911,E2 -4824.911} C_VEL
LIN {X 0,Y 523.941,Z 711.223,A -85,B 0,C 180,E1 -4827.679,E2 -4827.679} C_VEL
LIN {X 0,Y 523.957,Z 711.214,A -85,B 0,C 180,E1 -4830.677,E2 -4830.677} C_VEL
LIN {X 0,Y 523.977,Z 711.22,A -85,B 0,C 180,E1 -4833.729,E2 -4833.729} C_VEL
LIN {X 0,Y 523.915,Z 711.221,A -85,B 0,C 180,E1 -4836.27,E2 -4836.27} C_VEL
LIN {X 0,Y 523.948,Z 711.215,A -85,B 0,C 180,E1 -4838.767,E2 -4838.767} C_VEL
LIN {X 0,Y 523.951,Z 711.216,A -85,B 0,C 180,E1 -4841.221,E2 -4841.221} C_VEL
LIN {X 0,Y 523.935,Z 711.222,A -85,B 0,C 180,E1 -4843.639,E2 -4843.639} C_VEL
LIN {X 0,Y 523.941,Z 711.223,A -85,B 0,C 180,E1 -4846.028,E2 -4846.028} C_VEL
LIN {X 0,Y 524.016,Z 711.209,A -85,B 0,C 180,E1 -4848.394,E2 -4848.394} C_VEL
LIN {X 0,Y 524.003,Z 711.211,A -85,B 0,C 180,E1 -4851.516,E2 -4851.516} C_VEL
LIN {X 0,Y 524.082,Z 711.2,A -85,B 0,C 180,E1 -4854.614,E2 -4854.614} C_VEL
LIN {X 0,Y 524.113,Z 711.199,A -85,B 0,C 180,E1 -4857.695,E2 -4857.695} C_VEL
LIN {X 0,Y 524.12,Z 711.195,A -85,B 0,C 180,E1 -4860.768,E2 -4860.768} C_VEL
LIN {X 0,Y 524.041,Z 711.204,A -85,B 0,C 180,E1 -4863.075,E2 -4863.075} C_VEL
LIN {X 0,Y 524.026,Z 711.212,A -85,B 0,C 180,E1 -4866.159,E2 -4866.159} C_VEL
LIN {X 0,Y 523.988,Z 711.21,A -85,B 0,C 180,E1 -4869.262,E2 -4869.262} C_VEL
LIN {X 0,Y 524.002,Z 711.211,A -85,B 0,C 180,E1 -4871.737,E2 -4871.737} C_VEL
LIN {X 0,Y 523.99,Z 711.211,A -85,B 0,C 180,E1 -4875.05,E2 -4875.05} C_VEL
LIN {X 0,Y 523.947,Z 711.219,A -85,B 0,C 180,E1 -4877.97,E2 -4877.97} C_VEL
LIN {X 0,Y 523.975,Z 711.219,A -85,B 0,C 180,E1 -4880.41,E2 -4880.41} C_VEL
LIN {X 0,Y 523.912,Z 711.224,A -85,B 0,C 180,E1 -4882.894,E2 -4882.894} C_VEL
LIN {X 0,Y 523.899,Z 711.222,A -85,B 0,C 180,E1 -4885.422,E2 -4885.422} C_VEL
LIN {X 0,Y 523.916,Z 711.221,A -85,B 0,C 180,E1 -4888.002,E2 -4888.002} C_VEL
LIN {X 0,Y 523.937,Z 711.224,A -85,B 0,C 180,E1 -4890.853,E2 -4890.853} C_VEL
LIN {X 0,Y 523.929,Z 711.218,A -85,B 0,C 180,E1 -4893.729,E2 -4893.729} C_VEL
LIN {X 0,Y 523.89,Z 711.227,A -85,B 0,C 180,E1 -4896.399,E2 -4896.399} C_VEL
LIN {X 0,Y 523.909,Z 711.226,A -85,B 0,C 180,E1 -4899.086,E2 -4899.086} C_VEL
LIN {X 0,Y 523.895,Z 711.223,A -85,B 0,C 180,E1 -4902.125,E2 -4902.125} C_VEL
LIN {X 0,Y 523.936,Z 711.221,A -85,B 0,C 180,E1 -4905.311,E2 -4905.311} C_VEL
LIN {X 0,Y 523.879,Z 711.23,A -85,B 0,C 180,E1 -4906.891,E2 -4906.891} C_VEL
LIN {X 0,Y 523.199,Z 711.312,A -85,B 0,C 180,E1 -4907.532,E2 -4907.532} C_VEL
LIN {X 0,Y 520.357,Z 711.667,A -85,B 0,C 180,E1 -4908.574,E2 -4908.574} C_VEL
LIN {X 0,Y 517.965,Z 711.964,A -85,B 0,C 180,E1 -4909.413,E2 -4909.413} C_VEL
LIN {X 0,Y 516.941,Z 712.089,A -85,B 0,C 180,E1 -4910.061,E2 -4910.061} C_VEL
LIN {X 0,Y 516.859,Z 712.1,A -85,B 0,C 180,E1 -4910.28,E2 -4910.28} C_VEL
LIN {X 0,Y 516.817,Z 712.11,A -85,B 0,C 180,E1 -4913.249,E2 -4913.249} C_VEL
LIN {X 0,Y 516.869,Z 712.098,A -85,B 0,C 180,E1 -4916.118,E2 -4916.118} C_VEL
LIN {X 0,Y 516.851,Z 712.106,A -85,B 0,C 180,E1 -4918.944,E2 -4918.944} C_VEL
LIN {X 0,Y 516.843,Z 712.105,A -85,B 0,C 180,E1 -4921.58,E2 -4921.58} C_VEL
LIN {X 0,Y 516.842,Z 712.101,A -85,B 0,C 180,E1 -4924.206,E2 -4924.206} C_VEL
LIN {X 0,Y 516.858,Z 712.101,A -85,B 0,C 180,E1 -4926.776,E2 -4926.776} C_VEL
LIN {X 0,Y 516.942,Z 712.092,A -85,B 0,C 180,E1 -4929.732,E2 -4929.732} C_VEL
LIN {X 0,Y 516.887,Z 712.096,A -85,B 0,C 180,E1 -4932.595,E2 -4932.595} C_VEL
LIN {X 0,Y 516.936,Z 712.093,A -85,B 0,C 180,E1 -4935.03,E2 -4935.03} C_VEL
LIN {X 0,Y 516.929,Z 712.091,A -85,B 0,C 180,E1 -4938.233,E2 -4938.233} C_VEL
LIN {X 0,Y 516.921,Z 712.098,A -85,B 0,C 180,E1 -4941.399,E2 -4941.399} C_VEL
LIN {X 0,Y 516.983,Z 712.083,A -85,B 0,C 180,E1 -4944.54,E2 -4944.54} C_VEL
LIN {X 0,Y 517.075,Z 712.078,A -85,B 0,C 180,E1 -4947.663,E2 -4947.663} C_VEL
LIN {X 0,Y 517.068,Z 712.077,A -85,B 0,C 180,E1 -4950,E2 -4950} C_VEL
LIN {X 0,Y 517.076,Z 712.073,A -85,B 0,C 180,E1 -4952.337,E2 -4952.337} C_VEL
LIN {X 0,Y 516.978,Z 712.087,A -85,B 0,C 180,E1 -4956.244,E2 -4956.244} C_VEL
LIN {X 0,Y 516.94,Z 712.091,A -85,B 0,C 180,E1 -4959.39,E2 -4959.39} C_VEL
LIN {X 0,Y 516.956,Z 712.094,A -85,B 0,C 180,E1 -4961.807,E2 -4961.807} C_VEL
LIN {X 0,Y 516.949,Z 712.087,A -85,B 0,C 180,E1 -4965.146,E2 -4965.146} C_VEL
LIN {X 0,Y 516.917,Z 712.096,A -85,B 0,C 180,E1 -4968.223,E2 -4968.223} C_VEL
LIN {X 0,Y 516.917,Z 712.092,A -85,B 0,C 180,E1 -4970.702,E2 -4970.702} C_VEL
LIN {X 0,Y 516.89,Z 712.103,A -85,B 0,C 180,E1 -4974.073,E2 -4974.073} C_VEL
LIN {X 0,Y 516.853,Z 712.101,A -85,B 0,C 180,E1 -4976.662,E2 -4976.662} C_VEL
LIN {X 0,Y 516.913,Z 712.092,A -85,B 0,C 180,E1 -4979.523,E2 -4979.523} C_VEL
LIN {X 0,Y 516.898,Z 712.098,A -85,B 0,C 180,E1 -4982.543,E2 -4982.543} C_VEL
LIN {X 0,Y 516.869,Z 712.096,A -85,B 0,C 180,E1 -4985.33,E2 -4985.33} C_VEL
LIN {X 0,Y 516.884,Z 712.098,A -85,B 0,C 180,E1 -4987.943,E2 -4987.943} C_VEL
LIN {X 0,Y 516.887,Z 712.098,A -85,B 0,C 180,E1 -4990.742,E2 -4990.742} C_VEL
LIN {X 0,Y 516.886,Z 712.098,A -85,B 0,C 180,E1 -4992.832,E2 -4992.832} C_VEL
LIN {X 0,Y 516.899,Z 712.096,A -85,B 0,C 180,E1 -4995.007,E2 -4995.007} C_VEL
LIN {X 0,Y 516.921,Z 712.099,A -85,B 0,C 180,E1 -4998.398,E2 -4998.398} C_VEL
LIN {X 0,Y 516.927,Z 712.118,A -85,B 0,C 180,E1 -4998.897,E2 -4998.897} C_VEL
LIN {X 0,Y 518.365,Z 718.302,A -85,B 0,C 180,E1 -4999.228,E2 -4999.228} C_VEL
